(* IEC 61131-3 sources: SmartHomeNew/snapshots/2026-05-12, 47 files *)

(* ---- E_Heating_RootCause.dut ---- *)
TYPE E_Heating_RootCause :
(
    RC_NONE,
    RC_EMERGENCY_STOP,
    RC_GAS_SAFETY,
    RC_IO_OFFLINE,
    RC_BOILER_OFFLINE,
    RC_BOILER_ERROR,
    RC_NO_FLAME,
    RC_NO_FLOW,
    RC_PUMP_FAILURE,
    RC_VALVES_CLOSED,
    RC_NO_HEAT_TRANSFER,
    RC_LOW_SUPPLY_TEMP,
    RC_SENSOR_ERROR,
    RC_POLICY_BLOCKED,
    RC_UNKNOWN
);
END_TYPE

(* ---- E_Heating_Runtime_Phase.dut ---- *)
TYPE E_Heating_Runtime_Phase :
(
    HRP_DISABLED := 0,

    // Runtime startup / idle
    HRP_IDLE := 10,

    // Phase 1
    // DHW manager execution
    HRP_DHW := 20,

    // Phase 2
    // Heating runtime execution
    HRP_HEATING := 30,

    // Phase 3
    // Service and failsafe gating
    HRP_SERVICE_GATING := 40,

    // Phase 4
    // Runtime state publication
    HRP_STATE_PUBLICATION := 50,

    // Phase 5
    // Diagnostics / explainability
    HRP_DIAGNOSTICS := 60,

    // Phase 6
    // Output projection
    HRP_OUTPUT_PROJECTION := 70,

    // Runtime finished
    HRP_COMPLETE := 100,

    // Runtime error/fault state
    HRP_FAULT := 900
);
END_TYPE

(* ---- E_Modbus_RTU_RX_State.dut ---- *)
TYPE E_Modbus_RTU_RX_State :
(
    MB_RTU_RX_IDLE := 0,
    MB_RTU_RX_RECEIVING := 1,
    MB_RTU_RX_FRAME_READY := 2,
    MB_RTU_RX_CRC_ERROR := 3,
    MB_RTU_RX_OVERFLOW := 4,
    MB_RTU_RX_SHORT_FRAME := 5
);
END_TYPE

(* ---- E_System_Operating_Mode.dut ---- *)
TYPE E_System_Operating_Mode :
(
    MODE_NORMAL := 0,
    MODE_DEGRADED := 1,
    MODE_SAFE_STOP := 2,
    MODE_FREEZE_PROTECTION := 3
);
END_TYPE

(* ---- E_Trend_Parameter_Type.dut ---- *)
{attribute 'strict'}
TYPE E_Trend_Parameter_Type :
(
    TREND_PARAM_NONE := 0,
    TREND_PARAM_TEMP_AIR := 1,
    TREND_PARAM_TEMP_FLOOR := 2,
    TREND_PARAM_PRESSURE := 3,
    TREND_PARAM_PUMP_CURRENT := 4,
    TREND_PARAM_GAS_METHANE := 5,
    TREND_PARAM_GAS_CO := 6
) USINT;
END_TYPE

(* ---- ST_Device_Health.dut ---- *)
{attribute 'pack_mode' := '1'}
TYPE ST_Device_Health :
STRUCT
    Health_Score : BYTE := 100;
    Total_Runtime_Hours : UDINT;
    Starts_Count : UDINT;
    Last_Start_Current : REAL;
    Avg_Start_Current : REAL;
    Sample_Count : UDINT;
    Current_Sum : REAL;
    Maintenance_Required : BOOL;
    Warning_Message : STRING(50);
END_STRUCT
END_TYPE

(* ---- ST_FloorHeating_Circuit_Config.dut ---- *)
{attribute 'pack_mode' := '1'}
TYPE ST_FloorHeating_Circuit_Config :
STRUCT
    circuit_id : BYTE := 0;
    zone : BYTE := 0;
    manifold_id : BYTE := 1; // ID коллектора, к которому подключен контур
    sensor_id : BYTE := 1; // ID датчика температуры
    valve_id : BYTE := 1; // ID клапана
    control_type : BYTE := 1; // 0: по полу, 1: по воздуху
    design_temp : REAL := 35.0;
    min_temp : REAL := 20.0;
    max_temp : REAL := 45.0;
    pid_kp : REAL := 2.0;
    pwm_period_s : UINT := 600; // Период ШИМ в секундах (по умолчанию 10 минут)
END_STRUCT
END_TYPE

(* ---- ST_Heating_Runtime_Causality_Node.dut ---- *)
TYPE ST_Heating_Runtime_Causality_Node :
STRUCT
    // ======================================================
    // Node identity
    // ======================================================
    Node_ID : UINT;
    Node_Active : BOOL;

    // ======================================================
    // Runtime source state
    // ======================================================
    Runtime_Degraded : BOOL;
    Runtime_Fault : BOOL;

    // ======================================================
    // Cascade source state
    // ======================================================
    Cascade_Degraded : BOOL;
    Cascade_Boiler_Loss : BOOL;

    // ======================================================
    // OpenTherm source state
    // ======================================================
    OpenTherm_Degraded : BOOL;
    OpenTherm_Command_Invalid : BOOL;

    // ======================================================
    // Diagnostics source state
    // ======================================================
    Diagnostics_Degraded : BOOL;
    Explainability_Degraded : BOOL;

    // ======================================================
    // Sequencing/integrity state
    // ======================================================
    Sequencing_Invalid : BOOL;
    Ownership_Invalid : BOOL;
    Synchronization_Invalid : BOOL;

    // ======================================================
    // Causality severity
    // ======================================================
    Severity_Level : UINT;
    Root_Cause_Candidate : BOOL;

    // ======================================================
    // Node status
    // ======================================================
    Status_Code : UINT;
    Status_Text : STRING(128);
END_STRUCT
END_TYPE

(* ---- ST_Heating_Runtime_Execution_Frame.dut ---- *)
TYPE ST_Heating_Runtime_Execution_Frame :
STRUCT
    // ======================================================
    // Execution phase
    // ======================================================
    Phase : E_Heating_Runtime_Phase;

    // ======================================================
    // Execution lifecycle
    // ======================================================
    Frame_Started : BOOL;
    Frame_Completed : BOOL;
    Frame_Failed : BOOL;

    // ======================================================
    // Execution timing
    // ======================================================
    Frame_Start_MS : UDINT;
    Frame_End_MS : UDINT;
    Frame_Duration_MS : UDINT;

    // ======================================================
    // Execution integrity
    // ======================================================
    Sequencing_Valid : BOOL;
    Ownership_Valid : BOOL;
    Synchronization_Valid : BOOL;

    // ======================================================
    // Execution telemetry
    // ======================================================
    Runtime_Jitter_Detected : BOOL;
    Runtime_Latency_Detected : BOOL;
    Runtime_Degraded : BOOL;

    // ======================================================
    // Execution status
    // ======================================================
    Status_Code : UINT;
    Status_Text : STRING(128);
END_STRUCT
END_TYPE

(* ---- ST_Heating_Schedule_Event.dut ---- *)
{attribute 'pack_mode' := '1'}
TYPE ST_Heating_Schedule_Event :
STRUCT
    Enabled : BOOL := FALSE;
    Comfort_Time_MS : UDINT := 28800000; // 08:00 from midnight
    Weekday_Mask : BYTE := 127; // bit0=Mon ... bit6=Sun
    Preheat_Boost : REAL := 0.5;
    Adaptive_Enabled : BOOL := TRUE;
    Adaptive_Step_MS : UDINT := 300000; // 5 min
    Adaptive_Max_Offset_MS : UDINT := 3600000; // 60 min
END_STRUCT
END_TYPE

(* ---- ST_Modbus_RTU_Config.dut ---- *)
TYPE ST_Modbus_RTU_Config :
STRUCT
    Port_Name : STRING(32);
    Baudrate : UDINT;
    Parity : BYTE; // 0=None, 1=Even, 2=Odd
    Stop_Bits : BYTE; // 1 or 2
    Data_Bits : BYTE; // usually 8
    Slave_ID : BYTE;
    Poll_Interval_MS : UDINT;
    Request_Timeout_MS : UDINT;
    Retry_Count : INT;
END_STRUCT
END_TYPE

(* ---- ST_Modbus_RTU_Frame.dut ---- *)
TYPE ST_Modbus_RTU_Frame :
STRUCT
    Valid : BOOL;
    Length : UINT;
    Data : ARRAY[0..255] OF BYTE;
    CRC : WORD;
END_STRUCT
END_TYPE

(* ---- ST_OpenTherm_Register_Map.dut ---- *)
TYPE ST_OpenTherm_Register_Map :
STRUCT
    // Register offsets inside one boiler adapter block.
    // Real Modbus device addressing is configured by Base_Register + offsets.
    Base_Register : UINT;
    Cmd_Enable_Offset : UINT;
    Cmd_Setpoint_x10_Offset : UINT;
    Cmd_Seq_Lo_Offset : UINT;
    Cmd_Seq_Hi_Offset : UINT;

    Status_Heartbeat_Lo_Offset : UINT;
    Status_Heartbeat_Hi_Offset : UINT;
    Status_Ack_Seq_Lo_Offset : UINT;
    Status_Ack_Seq_Hi_Offset : UINT;
    Status_Word_Offset : UINT;
    Error_Code_Offset : UINT;
    Modulation_x10_Offset : UINT;
    Boiler_Temp_x10_Offset : UINT;
END_STRUCT
END_TYPE

(* ---- GVL_ACCESS_OUTPUT.gvl ---- *)
VAR_GLOBAL
    DO_Lock_1_Open : BOOL := FALSE;
    DO_Lock_1_Close : BOOL := FALSE;
    DO_Lock_2_Open : BOOL := FALSE;
    DO_Lock_2_Close : BOOL := FALSE;
    DO_Gate_Open : BOOL := FALSE;
    DO_Wicket_Open : BOOL := FALSE;
END_VAR

(* ---- GVL_DIAGNOSTICS_EXT.gvl ---- *)
{attribute 'qualified_only'}
VAR_GLOBAL
    // Health scores (0..1)
    G_Health_Heating : REAL := 1.0;
    G_Health_Safety : REAL := 1.0;
    G_Health_IO : REAL := 1.0;

    // Error counters
    G_Error_Count_Heating : UDINT := 0;
    G_Error_Count_Safety : UDINT := 0;
    G_Error_Count_IO : UDINT := 0;

    // Last error timestamps
    G_Last_Error_Time_Heating : UDINT := 0;
    G_Last_Error_Time_Safety : UDINT := 0;
    G_Last_Error_Time_IO : UDINT := 0;

    // Timing
    G_Last_Update_Time : UDINT := 0;

    // Cycle / watchdog statistics (interval between diagnostics executions)
    G_Cycle_Expected_MS : UDINT := 250;
    G_Cycle_Warning_MS : UDINT := 375;
    G_Cycle_Critical_MS : UDINT := 500;
    G_Cycle_Last_MS : UDINT := 0;
    G_Cycle_Max_MS : UDINT := 0;
    G_Cycle_Min_MS : UDINT := 0;
    G_Cycle_Avg_MS : REAL := 0.0;
    G_Cycle_Sample_Count : UDINT := 0;
    G_Cycle_Overrun_Count : UDINT := 0;
    G_Cycle_Critical_Count : UDINT := 0;
    G_Cycle_Last_Overrun_MS : UDINT := 0;
    G_Cycle_Last_Overrun_Time_MS : UDINT := 0;
    G_Cycle_Overrun_Active : BOOL := FALSE;
    G_Cycle_Critical_Active : BOOL := FALSE;

    // States
    G_Heating_State : INT := 0; // 0=OK,1=DEGRADED,2=CRITICAL
    G_Safety_State : INT := 0;
    G_IO_State : INT := 0;
END_VAR

(* ---- GVL_HEATING_REQUEST.gvl ---- *)
VAR_GLOBAL
    G_Freeze_Request : BOOL := FALSE;
    G_Target_Temperature : REAL := 0.0;
    G_Preheat_Request : BOOL := FALSE;
END_VAR

(* ---- GVL_INTENT_POLICY.gvl ---- *)
{attribute 'qualified_only'}
VAR_GLOBAL
    // Policy intent signals (NO logic, only transport)

    G_Preheat_Request : BOOL;
    G_Freeze_Request : BOOL;
    G_Eco_Mode_Request : BOOL;

    // Zone-level intents
    G_Zone_Heating_Request : ARRAY[1..GVL_CONSTANTS.C_MAX_ZONES] OF BOOL;
    G_Zone_Target_Adjustment : ARRAY[1..GVL_CONSTANTS.C_MAX_ZONES] OF REAL;

END_VAR

(* ---- GVL_SCENARIO_CONFIG.gvl ---- *)
{attribute 'qualified_only'}
VAR_GLOBAL
    // Scenario Engine configuration.
    // Used by PRG_Scenario_Engine only.

    G_Night_Start_Hour : INT := 22;
    G_Night_End_Hour : INT := 6;
    G_Access_Secure_Start_Hour : INT := 23;
    G_Access_Secure_End_Hour : INT := 5;

    G_Comfort_Base_Score : REAL := 10.0;
    G_Night_Base_Score : REAL := 40.0;
    G_Preheat_Base_Score : REAL := 50.0;
    G_VentBoost_Base_Score : REAL := 45.0;
    G_AccessSecure_Base_Score : REAL := 30.0;

    G_VentBoost_Humidity_Threshold : REAL := 65.0;

    G_Night_Activation_Threshold : INT := 30;
    G_Comfort_Activation_Threshold : INT := 40;
    G_VentBoost_Activation_Threshold : INT := 40;
    G_AccessSecure_Activation_Threshold : INT := 25;

    G_Fallback_Adapt_Confidence : REAL := 0.5;
    G_Fallback_Input_Confidence : REAL := 0.5;
END_VAR

(* ---- GVL_WATER_OUTPUT.gvl ---- *)
VAR_GLOBAL
    DO_Water_Valve_35_Close : BOOL := FALSE;
    DO_Water_Valve_36_Close : BOOL := FALSE;
    DO_Water_Zone_Enable : ARRAY[1..GVL_CONSTANTS.C_MAX_WATER_ZONES] OF BOOL;
END_VAR

(* ---- FB_Access_Control.st ---- *)
FUNCTION_BLOCK FB_Access_Control
VAR_INPUT
    VI_System_Time_MS   : UDINT; // Системное время (мс)
    VI_IsActivePLC      : BOOL; // Флаг: Данный ПЛК является ведущим (Active)
    VI_Armed            : BOOL; // Статус: Система безопасности находится под охраной
    VI_System_Mode      : E_System_Operating_Mode; // Агрегированный режим работы системы

    // Команды управления от HMI (через GVL_CONFIG)
    VI_Gate_Open_Req    : BOOL; // Запрос пользователя на открытие въездных ворот
    VI_Wicket_Open_Req  : BOOL; // Запрос пользователя на открытие калитки
    VI_Lock_1_Open_Req  : BOOL; // Запрос на разблокировку основного электрозамка дома
    VI_Lock_1_Close_Req : BOOL; // Запрос на блокировку основного электрозамка дома
    VI_Lock_2_Open_Req  : BOOL; // Запрос на разблокировку дополнительного электрозамка
    VI_Lock_2_Close_Req : BOOL; // Запрос на блокировку дополнительного электрозамка

    // Авторизация
    VI_PIN_Code         : STRING(4); // ПИН-код для авторизации
    VI_RFID_Tag         : STRING(20); // RFID/NFC метка для авторизации

    // Настройки из конфигурации безопасности (длительности импульсов)
    VI_Config           : ST_Security_Global_Config;
END_VAR
VAR_IN_OUT
    VI_Access_Codes     : ARRAY[1..GVL_CONSTANTS.C_MAX_ACCESS_CODES] OF DWORD;
    VI_RFID_Tags        : ARRAY[1..GVL_CONSTANTS.C_MAX_ACCESS_CODES] OF STRING(20);
END_VAR
VAR_OUTPUT
    VO_Gate_Open        : BOOL; // Выход: Импульс на открытие ворот (сухой контакт)
    VO_Wicket_Open      : BOOL; // Выход: Импульс на открытие калитки (электрозащелка)
    VO_Lock_1_Open      : BOOL; // Выход: Импульс на разблокировку замка №1
    VO_Lock_1_Close     : BOOL; // Выход: Импульс на блокировку замка №1
    VO_Lock_2_Open      : BOOL; // Выход: Импульс на разблокировку замка №2
    VO_Lock_2_Close     : BOOL; // Выход: Импульс на блокировку замка №2
END_VAR
VAR
    // Таймеры для формирования импульсов управления заданной длительности
    L_Gate_Timer        : TP; // Таймер импульса ворот
    L_Wicket_Timer      : TP; // Таймер импульса калитки
    L_Lock_1_Open_T     : TP; // Таймер открытия замка №1
    L_Lock_1_Close_T    : TP; // Таймер закрытия замка №1
    L_Lock_2_Open_T     : TP; // Таймер открытия замка №2
    L_Lock_2_Close_T    : TP; // Таймер закрытия замка №2

    L_Prev_Armed        : BOOL; // Предыдущее состояние охраны (для детекции фронта постановки)
    L_Auto_Lock_Req     : BOOL; // Флаг автоматического закрытия всех замков при постановке на охрану

    R_Trig_Gate         : R_TRIG;
    R_Trig_Wicket       : R_TRIG;
    R_Trig_Lock_1_O     : R_TRIG;
    R_Trig_Lock_1_C     : R_TRIG;
    R_Trig_Lock_2_O     : R_TRIG;
    R_Trig_Lock_2_C     : R_TRIG;

    fbAccessCode        : FB_AccessCode_Manager;
    L_Valid_PIN         : BOOL;
END_VAR

// Если ПЛК находится в режиме Standby (резерв), он не должен управлять выходами
IF NOT VI_IsActivePLC THEN
    RETURN;
END_IF;

IF VI_System_Mode = E_System_Operating_Mode.MODE_SAFE_STOP THEN
    VO_Gate_Open := FALSE;
    VO_Wicket_Open := FALSE;
    VO_Lock_1_Open := FALSE;
    VO_Lock_2_Open := FALSE;
    RETURN;
END_IF;

// 1. Логика автоматического закрытия замков при постановке на охрану (ТЗ 3.0)
// При переходе системы в режим "Охрана" принудительно блокируем все замки
IF VI_Armed AND NOT L_Prev_Armed THEN
    L_Auto_Lock_Req := TRUE;
END_IF;
L_Prev_Armed := VI_Armed;

// Детекторы фронта для команд
R_Trig_Gate(CLK := VI_Gate_Open_Req);
R_Trig_Wicket(CLK := VI_Wicket_Open_Req);
R_Trig_Lock_1_O(CLK := VI_Lock_1_Open_Req);
R_Trig_Lock_1_C(CLK := VI_Lock_1_Close_Req OR L_Auto_Lock_Req);
R_Trig_Lock_2_O(CLK := VI_Lock_2_Open_Req);
R_Trig_Lock_2_C(CLK := VI_Lock_2_Close_Req OR L_Auto_Lock_Req);

// Проверка PIN-кода или RFID-метки через менеджер кодов
fbAccessCode(
    VI_System_Time_MS := VI_System_Time_MS,
    VI_IsActivePLC := VI_IsActivePLC,
    VI_Code_To_Check := VI_PIN_Code,
    VI_RFID_To_Check := VI_RFID_Tag,
    VI_Access_Codes := VI_Access_Codes,
    VI_RFID_Tags := VI_RFID_Tags,
    VO_Code_Valid => L_Valid_PIN
);

// 2. Формирование импульсов управления исполнительными механизмами (Pulse Control)
// Открытие ворот и калитки требует валидного ПИН-кода или RFID-метки, если система под охраной
L_Gate_Timer(IN := R_Trig_Gate.Q AND (NOT VI_Armed OR L_Valid_PIN), PT := TO_TIME(VI_Config.gate_open_pulse_ms));
VO_Gate_Open := L_Gate_Timer.Q;

L_Wicket_Timer(IN := R_Trig_Wicket.Q AND (NOT VI_Armed OR L_Valid_PIN), PT := TO_TIME(VI_Config.wicket_open_pulse_ms));
VO_Wicket_Open := L_Wicket_Timer.Q;

L_Lock_1_Open_T(IN := R_Trig_Lock_1_O.Q AND (NOT VI_Armed OR L_Valid_PIN), PT := TO_TIME(VI_Config.lock_open_pulse_ms));
VO_Lock_1_Open := L_Lock_1_Open_T.Q;

L_Lock_1_Close_T(IN := R_Trig_Lock_1_C.Q, PT := TO_TIME(VI_Config.lock_close_pulse_ms));
VO_Lock_1_Close := L_Lock_1_Close_T.Q;

L_Lock_2_Open_T(IN := R_Trig_Lock_2_O.Q AND (NOT VI_Armed OR L_Valid_PIN), PT := TO_TIME(VI_Config.lock_open_pulse_ms));
VO_Lock_2_Open := L_Lock_2_Open_T.Q;

L_Lock_2_Close_T(IN := R_Trig_Lock_2_C.Q, PT := TO_TIME(VI_Config.lock_close_pulse_ms));
VO_Lock_2_Close := L_Lock_2_Close_T.Q;

// Сброс флага автоматического закрытия
IF L_Auto_Lock_Req THEN
    L_Auto_Lock_Req := FALSE;
END_IF;
// >>> BULK_SYNC_ANCHOR: FB_Access_Control <<<
END_FUNCTION_BLOCK

(* ---- FB_AccessCode_Manager.st ---- *)
FUNCTION_BLOCK FB_AccessCode_Manager
VAR_INPUT
    VI_System_Time_MS : UDINT;
    VI_IsActivePLC    : BOOL;
    VI_Code_To_Check  : STRING(4);
    VI_RFID_To_Check  : STRING(20);
END_VAR
VAR_IN_OUT
    VI_Access_Codes   : ARRAY[1..GVL_CONSTANTS.C_MAX_ACCESS_CODES] OF DWORD;
    VI_RFID_Tags      : ARRAY[1..GVL_CONSTANTS.C_MAX_ACCESS_CODES] OF STRING(20);
END_VAR
VAR_OUTPUT
    VO_Code_Valid     : BOOL;
END_VAR
VAR
    L_i : INT;
    pCode : POINTER TO BYTE;
    L_CRC_Calc : FB_CRC32_Calculator;
    L_Input_Hash : DWORD;
END_VAR

VO_Code_Valid := FALSE;

// Вычисляем хэш введенного кода
IF LEN(VI_Code_To_Check) > 0 THEN
    pCode := ADR(VI_Code_To_Check);
    L_Input_Hash := 0;
    FOR L_i := 1 TO GVL_CONSTANTS.C_MAX_ACCESS_CODES DO
        IF VI_Access_Codes[L_i] <> 0 AND VI_Access_Codes[L_i] = L_Input_Hash THEN
            VO_Code_Valid := TRUE;
            RETURN;
        END_IF;
    END_FOR;
END_IF;

// Проверяем RFID метку
IF LEN(VI_RFID_To_Check) > 0 THEN
    FOR L_i := 1 TO GVL_CONSTANTS.C_MAX_ACCESS_CODES DO
        IF VI_RFID_Tags[L_i] <> '' AND VI_RFID_Tags[L_i] = VI_RFID_To_Check THEN
            VO_Code_Valid := TRUE;
            RETURN;
        END_IF;
    END_FOR;
END_IF;
// >>> BULK_SYNC_ANCHOR: FB_AccessCode_Manager <<<
END_FUNCTION_BLOCK

(* ---- FB_Command_Deduplication.st ---- *)
FUNCTION_BLOCK FB_Command_Deduplication
VAR_INPUT
    VI_Command_ID : UDINT; // Unique ID from Gateway/HMI
    VI_Command_Type : E_Gateway_Command_Type;
    VI_Command_Value : REAL;
    VI_System_Time_MS : UDINT;
END_VAR
VAR_OUTPUT
    VO_Is_New_Command : BOOL; // TRUE if this command should be executed
    VO_Processed_ID : UDINT;
END_VAR
VAR
    L_Processed_History : ARRAY[0..GVL_CONSTANTS.C_MAX_DEDUPLICATION_HISTORY-1] OF UDINT; // Ring buffer of last processed IDs
    L_Processed_Times   : ARRAY[0..GVL_CONSTANTS.C_MAX_DEDUPLICATION_HISTORY-1] OF UDINT; // Timestamps for processed IDs
    L_History_Index : INT := 0;
    L_i : INT;
    L_Found : BOOL;
END_VAR

// Check if command ID is already in history
L_Found := FALSE;
FOR L_i := 0 TO GVL_CONSTANTS.C_MAX_DEDUPLICATION_HISTORY-1 DO
    IF L_Processed_History[L_i] = VI_Command_ID AND VI_Command_ID <> 0 THEN
        // Check if the command is not too old (e.g., 1 hour = 3600000 ms)
        IF (VI_System_Time_MS - L_Processed_Times[L_i]) < 3600000 THEN
            L_Found := TRUE;
            EXIT;
        END_IF;
    END_IF;
END_FOR;

IF NOT L_Found AND VI_Command_ID <> 0 THEN
    // New command detected
    VO_Is_New_Command := TRUE;
    VO_Processed_ID := VI_Command_ID;

    // Add to history
    L_Processed_History[L_History_Index] := VI_Command_ID;
    L_Processed_Times[L_History_Index] := VI_System_Time_MS;
    L_History_Index := L_History_Index + 1;
    IF L_History_Index > GVL_CONSTANTS.C_MAX_DEDUPLICATION_HISTORY-1 THEN
        L_History_Index := 0;
    END_IF;
ELSE
    // Duplicate or empty command
    VO_Is_New_Command := FALSE;
    VO_Processed_ID := 0;
END_IF;
END_FUNCTION_BLOCK

(* ---- FB_Heating_Adaptive_Target.st ---- *)
// ==============================================================================
// Adaptive target calculation for heating supply temperature
// ==============================================================================
FUNCTION_BLOCK FB_Heating_Adaptive_Target
VAR_INPUT
    VI_Base_Target_Supply_Temp : REAL;
    VI_Global_Target_Temperature : REAL;
END_VAR

VAR_IN_OUT
    VI_Zone_Configs : ARRAY[1..GVL_CONSTANTS.C_MAX_HEATING_CIRCUITS] OF ST_FloorHeating_Circuit_Config;
    VI_Floor_Temps : ARRAY[1..GVL_CONSTANTS.C_MAX_HEATING_CIRCUITS] OF REAL;
    VI_Room_Temps : ARRAY[1..GVL_CONSTANTS.C_MAX_ZONES] OF REAL;
END_VAR

VAR_OUTPUT
    VO_Target_Supply_Temp : REAL;
    VO_Adaptive_Correction : REAL;
    VO_Adaptive_Effective_Delta : REAL;
    VO_Adaptive_Max_Delta : REAL;
END_VAR

VAR
    L_Adaptive_Zone_i : INT;
    L_Zone_Index : INT;
    L_Adaptive_Delta : REAL;
    L_Adaptive_Weighted_Sum : REAL;
    L_Adaptive_Weight_Total : REAL;
    L_Adaptive_Weight : REAL;
END_VAR

VO_Target_Supply_Temp := VI_Base_Target_Supply_Temp;
VO_Adaptive_Max_Delta := 0.0;
L_Adaptive_Weighted_Sum := 0.0;
L_Adaptive_Weight_Total := 0.0;
VO_Adaptive_Effective_Delta := 0.0;
VO_Adaptive_Correction := 0.0;

IF VI_Global_Target_Temperature > 0.0 THEN
    VO_Target_Supply_Temp := VI_Global_Target_Temperature;
END_IF;

FOR L_Adaptive_Zone_i := 1 TO GVL_CONSTANTS.C_MAX_HEATING_CIRCUITS DO
    L_Zone_Index := VI_Zone_Configs[L_Adaptive_Zone_i].zone;

    IF (L_Zone_Index >= 1) AND (L_Zone_Index <= GVL_CONSTANTS.C_MAX_ZONES) THEN
        CASE VI_Zone_Configs[L_Adaptive_Zone_i].control_type OF
            0:
                L_Adaptive_Delta :=
                    VI_Zone_Configs[L_Adaptive_Zone_i].design_temp -
                    VI_Floor_Temps[L_Adaptive_Zone_i];
                L_Adaptive_Weight := 0.6;
            1, 2:
                L_Adaptive_Delta :=
                    VI_Zone_Configs[L_Adaptive_Zone_i].design_temp -
                    VI_Room_Temps[L_Zone_Index];
                L_Adaptive_Weight := 1.0;
            ELSE
                L_Adaptive_Delta :=
                    VI_Zone_Configs[L_Adaptive_Zone_i].design_temp -
                    VI_Room_Temps[L_Zone_Index];
                L_Adaptive_Weight := 0.8;
        END_CASE;

        IF L_Zone_Index <= 4 THEN
            L_Adaptive_Weight := L_Adaptive_Weight * 1.2;
        ELSIF L_Zone_Index >= 9 THEN
            L_Adaptive_Weight := L_Adaptive_Weight * 0.7;
        END_IF;

        IF L_Adaptive_Weight > 2.0 THEN
            L_Adaptive_Weight := 2.0;
        ELSIF L_Adaptive_Weight < 0.2 THEN
            L_Adaptive_Weight := 0.2;
        END_IF;

        IF L_Adaptive_Delta > VO_Adaptive_Max_Delta THEN
            VO_Adaptive_Max_Delta := L_Adaptive_Delta;
        END_IF;

        L_Adaptive_Weighted_Sum := L_Adaptive_Weighted_Sum + (L_Adaptive_Delta * L_Adaptive_Weight);
        L_Adaptive_Weight_Total := L_Adaptive_Weight_Total + L_Adaptive_Weight;
    END_IF;
END_FOR;

IF L_Adaptive_Weight_Total > 0.0 THEN
    VO_Adaptive_Effective_Delta := L_Adaptive_Weighted_Sum / L_Adaptive_Weight_Total;
END_IF;

IF VO_Adaptive_Effective_Delta > 1.5 THEN
    VO_Adaptive_Correction := 2.0;
ELSIF VO_Adaptive_Effective_Delta > 0.7 THEN
    VO_Adaptive_Correction := 1.0;
ELSIF VO_Adaptive_Effective_Delta < -1.5 THEN
    VO_Adaptive_Correction := -2.0;
ELSIF VO_Adaptive_Effective_Delta < -0.7 THEN
    VO_Adaptive_Correction := -1.0;
ELSE
    VO_Adaptive_Correction := 0.0;
END_IF;

IF VO_Adaptive_Max_Delta > 2.5 AND VO_Adaptive_Correction < 2.0 THEN
    VO_Adaptive_Correction := 2.0;
END_IF;

VO_Target_Supply_Temp := VO_Target_Supply_Temp + VO_Adaptive_Correction;

IF VO_Target_Supply_Temp < 20.0 THEN
    VO_Target_Supply_Temp := 20.0;
ELSIF VO_Target_Supply_Temp > 45.0 THEN
    VO_Target_Supply_Temp := 45.0;
END_IF;

// >>> BULK_SYNC_ANCHOR: FB_Heating_Adaptive_Target <<<
END_FUNCTION_BLOCK

(* ---- FB_Heating_Allocation_Filter.st ---- *)
// ==============================================================================
// Heating allocation filter
// Runtime decision gate between Demand_Map and Manifold_Control.
//
// IMPORTANT:
// This FB is NOT a second runtime owner.
// This FB is NOT an orchestration layer.
//
// Actual ownership remains in:
// PRG_Heating
// → FB_Heating_System_Manager
// → active subsystem owners.
//
// Current responsibility:
// - manifold availability gating;
// - service-state filtering;
// - freeze-mode exceptions;
// - bounded demand authorization.
//
// Optional responsibility when explicitly enabled:
// - priority-based allocation;
// - thermal budget limiting.
// ==============================================================================
FUNCTION_BLOCK FB_Heating_Allocation_Filter
VAR_INPUT
    // Master runtime enable.
    // FALSE = strict passthrough.
    VI_Enable : BOOL;

    // Optional policy layer.
    // FALSE = only availability/service/degraded gate is active.
    VI_Enable_Policy_Allocation : BOOL := FALSE;

    // System-level context.
    VI_Freeze_Mode_Active : BOOL;
    VI_DHW_Heating_Demand : BOOL;

    // Current manifold demand.
    VI_Manifold_Demand_Map : ARRAY[1..GVL_CONSTANTS.C_MAX_MANIFOLDS] OF BOOL;

    // Runtime/service availability.
    VI_Manifold_Available : ARRAY[1..GVL_CONSTANTS.C_MAX_MANIFOLDS] OF BOOL;
    VI_Manifold_In_Service : ARRAY[1..GVL_CONSTANTS.C_MAX_MANIFOLDS] OF BOOL;
    VI_Manifold_Subsystem_Degraded : ARRAY[1..GVL_CONSTANTS.C_MAX_MANIFOLDS] OF BOOL;

    // Policy inputs from active configuration.
    VI_Manifold_Base_Priority : ARRAY[1..GVL_CONSTANTS.C_MAX_MANIFOLDS] OF INT;
    VI_Manifold_Thermal_Weight : ARRAY[1..GVL_CONSTANTS.C_MAX_MANIFOLDS] OF REAL;
    VI_Max_Thermal_Budget : REAL := REAL#0.0;
END_VAR
VAR_OUTPUT
    // Authorized demand.
    VO_Manifold_Demand_Filtered : ARRAY[1..GVL_CONSTANTS.C_MAX_MANIFOLDS] OF BOOL;

    // Runtime degraded indicator.
    VO_Allocation_Degraded : BOOL;

    // Explainability/diagnostics.
    VO_Manifold_Allowed : ARRAY[1..GVL_CONSTANTS.C_MAX_MANIFOLDS] OF BOOL;
    VO_Manifold_Block_Reason : ARRAY[1..GVL_CONSTANTS.C_MAX_MANIFOLDS] OF E_Heating_Allocation_Block_Reason;

    // Policy diagnostics.
    VO_Manifold_Priority_Effective : ARRAY[1..GVL_CONSTANTS.C_MAX_MANIFOLDS] OF INT;
    VO_Thermal_Budget_Used : REAL;
END_VAR
VAR
    L_i : INT;
    L_CurrentPriority : INT;
    L_MaxPriority : INT;
    L_Used : REAL;
    L_Weight : REAL;
    L_AnyPolicyBlock : BOOL;
END_VAR

// ======================================================
// DEFAULT STATE
// ======================================================
VO_Allocation_Degraded := FALSE;
VO_Thermal_Budget_Used := REAL#0.0;
L_AnyPolicyBlock := FALSE;

FOR L_i := 1 TO GVL_CONSTANTS.C_MAX_MANIFOLDS DO
    VO_Manifold_Demand_Filtered[L_i] := VI_Manifold_Demand_Map[L_i];
    VO_Manifold_Allowed[L_i] := TRUE;
    VO_Manifold_Block_Reason[L_i] := E_Heating_Allocation_Block_Reason.NONE;
    VO_Manifold_Priority_Effective[L_i] := VI_Manifold_Base_Priority[L_i];
END_FOR;

// ======================================================
// STRICT PASSTHROUGH MODE
// ======================================================
IF NOT VI_Enable THEN
    RETURN;
END_IF;

// ======================================================
// FREEZE EXCEPTION MODE
//
// Freeze protection has higher authority than
// service gating and policy throttling.
// ======================================================
IF VI_Freeze_Mode_Active THEN
    FOR L_i := 1 TO GVL_CONSTANTS.C_MAX_MANIFOLDS DO
        IF VI_Manifold_Demand_Map[L_i] THEN
            VO_Manifold_Block_Reason[L_i] := E_Heating_Allocation_Block_Reason.FREEZE_BYPASS;
        END_IF;
    END_FOR;
    RETURN;
END_IF;

// ======================================================
// DHW PRIORITY GATE
//
// Manifold_Control already owns DHW shutdown.
// Keep this filter transparent during DHW hold to avoid
// creating duplicate DHW authority here.
// ======================================================
IF VI_DHW_Heating_Demand THEN
    FOR L_i := 1 TO GVL_CONSTANTS.C_MAX_MANIFOLDS DO
        IF VI_Manifold_Demand_Map[L_i] THEN
            VO_Manifold_Block_Reason[L_i] := E_Heating_Allocation_Block_Reason.DHW_BYPASS;
        END_IF;
    END_FOR;
    RETURN;
END_IF;

// ======================================================
// MANIFOLD AUTHORIZATION FILTER
// ======================================================
FOR L_i := 1 TO GVL_CONSTANTS.C_MAX_MANIFOLDS DO

    IF NOT VI_Manifold_Available[L_i] THEN
        VO_Manifold_Allowed[L_i] := FALSE;
        VO_Manifold_Block_Reason[L_i] := E_Heating_Allocation_Block_Reason.PRESSURE_UNAVAILABLE;
    END_IF;

    IF NOT VI_Manifold_In_Service[L_i] THEN
        VO_Manifold_Allowed[L_i] := FALSE;
        VO_Manifold_Block_Reason[L_i] := E_Heating_Allocation_Block_Reason.SERVICE_DISABLED;
    END_IF;

    IF VI_Manifold_Subsystem_Degraded[L_i] THEN
        VO_Manifold_Allowed[L_i] := FALSE;
        VO_Manifold_Block_Reason[L_i] := E_Heating_Allocation_Block_Reason.PREDICTIVE_DEGRADED;
    END_IF;

    IF VI_Manifold_Demand_Map[L_i] AND NOT VO_Manifold_Allowed[L_i] THEN
        VO_Manifold_Demand_Filtered[L_i] := FALSE;
        VO_Allocation_Degraded := TRUE;
    END_IF;

END_FOR;

// ======================================================
// OPTIONAL POLICY LAYER
//
// This layer can only reduce demand that is already
// authorized by availability/service/degraded checks.
// It never creates new demand and never writes outputs.
// ======================================================
IF NOT VI_Enable_Policy_Allocation THEN
    RETURN;
END_IF;

// Invalid or unset budget means no policy throttling.
IF VI_Max_Thermal_Budget <= REAL#0.0 THEN
    RETURN;
END_IF;

// Rebuild output demand from allowed candidates only.
FOR L_i := 1 TO GVL_CONSTANTS.C_MAX_MANIFOLDS DO
    VO_Manifold_Demand_Filtered[L_i] := FALSE;
END_FOR;

L_MaxPriority := 0;
FOR L_i := 1 TO GVL_CONSTANTS.C_MAX_MANIFOLDS DO
    IF VI_Manifold_Demand_Map[L_i] AND VO_Manifold_Allowed[L_i] THEN
        IF VO_Manifold_Priority_Effective[L_i] > L_MaxPriority THEN
            L_MaxPriority := VO_Manifold_Priority_Effective[L_i];
        END_IF;
    END_IF;
END_FOR;

L_Used := REAL#0.0;

FOR L_CurrentPriority := L_MaxPriority TO 0 BY -1 DO
    FOR L_i := 1 TO GVL_CONSTANTS.C_MAX_MANIFOLDS DO
        IF VI_Manifold_Demand_Map[L_i]
           AND VO_Manifold_Allowed[L_i]
           AND (VO_Manifold_Priority_Effective[L_i] = L_CurrentPriority) THEN

            L_Weight := VI_Manifold_Thermal_Weight[L_i];
            IF L_Weight <= REAL#0.0 THEN
                L_Weight := REAL#1.0;
            END_IF;

            IF (L_Used + L_Weight) <= VI_Max_Thermal_Budget THEN
                VO_Manifold_Demand_Filtered[L_i] := TRUE;
                L_Used := L_Used + L_Weight;
            ELSE
                L_AnyPolicyBlock := TRUE;
                IF VO_Manifold_Block_Reason[L_i] = E_Heating_Allocation_Block_Reason.NONE THEN
                    VO_Manifold_Block_Reason[L_i] := E_Heating_Allocation_Block_Reason.POLICY_BUDGET_SHED;
                END_IF;
            END_IF;
        END_IF;
    END_FOR;
END_FOR;

VO_Thermal_Budget_Used := L_Used;

IF L_AnyPolicyBlock THEN
    VO_Allocation_Degraded := TRUE;
END_IF;

END_FUNCTION_BLOCK
// >>> BULK_SYNC_ANCHOR: FB_Heating_Allocation_Filter <<<

(* ---- FB_Heating_Boiler_Control.st ---- *)
// ==============================================================================
// Heating boiler control helper
// ==============================================================================
FUNCTION_BLOCK FB_Heating_Boiler_Control
VAR_INPUT
    VI_System_Time_MS : UDINT;
    VI_IsActivePLC : BOOL;
    VI_DHW_Heating_Demand : BOOL;
    VI_DHW_Target_Temp : REAL;
    VI_Target_Supply_Temp : REAL;
    VI_Freeze_Mode_Active : BOOL;
    VI_Policy_Degraded : BOOL;
    VI_Manifold_Pumps : ARRAY[1..GVL_CONSTANTS.C_MAX_MANIFOLDS] OF BOOL;
    VI_Manifold_Valves : ARRAY[1..GVL_CONSTANTS.C_MAX_MANIFOLDS] OF REAL;
    VI_Boiler_Flame_Status : ARRAY[1..GVL_CONSTANTS.C_MAX_BOILERS] OF BOOL;
    VI_Boiler_Error_Status : ARRAY[1..GVL_CONSTANTS.C_MAX_BOILERS] OF BOOL;
    VI_Boiler_OT_Online : ARRAY[1..GVL_CONSTANTS.C_MAX_BOILERS] OF BOOL;
END_VAR
VAR_IN_OUT
    VI_Boiler_Modulation : ARRAY[1..GVL_CONSTANTS.C_MAX_BOILERS] OF REAL;
END_VAR
VAR_OUTPUT
    VO_Boiler_OT_Enable : ARRAY[1..GVL_CONSTANTS.C_MAX_BOILERS] OF BOOL;
    VO_Boiler_OT_Setpoint : ARRAY[1..GVL_CONSTANTS.C_MAX_BOILERS] OF REAL;
    VO_Boiler_Status : ARRAY[1..GVL_CONSTANTS.C_MAX_BOILERS] OF ST_Boiler_Status;
    VO_Any_Subsystem_Degraded : BOOL;
    VO_Lead_Boiler : BYTE;
    VO_Demand_Power : REAL;
END_VAR
VAR
    L_i : INT;
    L_Delta_MS : UDINT;
    L_Last_Scan_Time : UDINT;
    L_Scan_Time_Init : BOOL := FALSE;
    L_Boiler_Request_Enable : ARRAY[1..GVL_CONSTANTS.C_MAX_BOILERS] OF BOOL;
    L_Boiler_Request_Setpoint : ARRAY[1..GVL_CONSTANTS.C_MAX_BOILERS] OF REAL;
    L_Boiler_OT_Command_Valid : ARRAY[1..GVL_CONSTANTS.C_MAX_BOILERS] OF BOOL;
    L_Transport_Degraded : BOOL;
    L_Available_Count : UINT;
    L_Active_Count : UINT;
    L_Any_Transport_Degraded : BOOL;
    L_Any_Ignition_Timeout : BOOL;
    L_Any_Flame : BOOL;
    L_Boiler_Life : ARRAY[1..GVL_CONSTANTS.C_MAX_BOILERS] OF FB_Lifetime_Predictor;
    fbBoilerCascade : FB_Boiler_Cascade_Manager;
    fbBoilerOpenTherm : FB_Boiler_OpenTherm_Interface;
END_VAR

VO_Any_Subsystem_Degraded := FALSE;
VO_Demand_Power := 0.0;

L_Available_Count := 0;
L_Active_Count := 0;
L_Any_Transport_Degraded := FALSE;
L_Any_Ignition_Timeout := FALSE;
L_Any_Flame := FALSE;

FOR L_i := 1 TO GVL_CONSTANTS.C_MAX_MANIFOLDS DO
    IF VI_Manifold_Pumps[L_i] THEN
        VO_Demand_Power := VO_Demand_Power + VI_Manifold_Valves[L_i];
    END_IF;
END_FOR;

IF VI_Freeze_Mode_Active AND VO_Demand_Power < 20.0 THEN
    VO_Demand_Power := 20.0;
END_IF;

IF VI_Policy_Degraded THEN
    IF VO_Demand_Power > 60.0 THEN
        VO_Demand_Power := 60.0;
    END_IF;
END_IF;

fbBoilerCascade(
    VI_Enable := VI_IsActivePLC AND ((VO_Demand_Power > GVL_CONSTANTS.C_BOILER_CASCADE_MIN_DEMAND) OR VI_Freeze_Mode_Active OR VI_DHW_Heating_Demand),
    VI_System_Time_MS := VI_System_Time_MS,
    VI_Boiler_Stop := FALSE,
    VI_DHW_Heating_Demand := VI_DHW_Heating_Demand,
    VI_DHW_Target_Temp := VI_DHW_Target_Temp,
    VI_Target_Supply_Temp := VI_Target_Supply_Temp,
    VI_Demand_Power := VO_Demand_Power,
    VI_Boiler_Flame_Status := VI_Boiler_Flame_Status,
    VI_Boiler_Error_Status := VI_Boiler_Error_Status,
    VI_Boiler_OT_Online := VI_Boiler_OT_Online,
    VI_Boiler_Modulation := VI_Boiler_Modulation,
    VO_Boiler_Enable => L_Boiler_Request_Enable,
    VO_Boiler_Setpoint => L_Boiler_Request_Setpoint,
    VO_Lead_Boiler => VO_Lead_Boiler
);

FOR L_i := 1 TO GVL_CONSTANTS.C_MAX_BOILERS DO
    IF L_Boiler_Request_Enable[L_i] THEN
        L_Boiler_Request_Setpoint[L_i] := LIMIT(
            GVL_CONSTANTS.C_BOILER_SETPOINT_MIN,
            L_Boiler_Request_Setpoint[L_i],
            80.0
        );
    END_IF;
END_FOR;

FOR L_i := 1 TO GVL_CONSTANTS.C_MAX_BOILERS DO
    IF NOT VI_Boiler_OT_Online[L_i] OR VI_Boiler_Error_Status[L_i] THEN
        L_Boiler_Request_Enable[L_i] := FALSE;
        L_Boiler_Request_Setpoint[L_i] := 0.0;
    END_IF;
END_FOR;

fbBoilerOpenTherm(
    VI_Enable := L_Boiler_Request_Enable,
    VI_Setpoint := L_Boiler_Request_Setpoint,
    VI_OT_Online := VI_Boiler_OT_Online,
    VI_OT_Error := VI_Boiler_Error_Status,
    VO_OT_Enable => VO_Boiler_OT_Enable,
    VO_OT_Setpoint => VO_Boiler_OT_Setpoint,
    VO_OT_Command_Valid => L_Boiler_OT_Command_Valid
);

FOR L_i := 1 TO GVL_CONSTANTS.C_MAX_BOILERS DO

    L_Transport_Degraded :=
        L_Boiler_Request_Enable[L_i] AND
        (
            NOT L_Boiler_OT_Command_Valid[L_i] OR
            NOT VI_Boiler_OT_Online[L_i] OR
            VI_Boiler_Error_Status[L_i]
        );

    VO_Boiler_Status[L_i].OT_Online := VI_Boiler_OT_Online[L_i];
    VO_Boiler_Status[L_i].OT_Command_Valid := L_Boiler_OT_Command_Valid[L_i];
    VO_Boiler_Status[L_i].OT_Transport_Degraded := L_Transport_Degraded;
    VO_Boiler_Status[L_i].OT_Adapter_Error :=
        GVL_OPENTHERM_ADAPTER.G_Status[L_i].Adapter_Error;

    VO_Boiler_Status[L_i].Active := L_Boiler_Request_Enable[L_i];
    VO_Boiler_Status[L_i].Running := VI_Boiler_Flame_Status[L_i];
    VO_Boiler_Status[L_i].Warning := L_Transport_Degraded;
    VO_Boiler_Status[L_i].Error := VI_Boiler_Error_Status[L_i];

    VO_Boiler_Status[L_i].Available :=
        VI_Boiler_OT_Online[L_i] AND
        NOT VI_Boiler_Error_Status[L_i] AND
        NOT L_Transport_Degraded;

    VO_Boiler_Status[L_i].Selected_By_Cascade :=
        L_Boiler_Request_Enable[L_i];

    VO_Boiler_Status[L_i].Transport_Missing :=
        NOT VI_Boiler_OT_Online[L_i];

    VO_Boiler_Status[L_i].Flame_Missing :=
        L_Boiler_Request_Enable[L_i] AND
        NOT VI_Boiler_Flame_Status[L_i] AND
        NOT L_Transport_Degraded;

    VO_Boiler_Status[L_i].Ignition_Timeout :=
        VO_Boiler_Status[L_i].Flame_Missing AND
        (GVL_STATE.G_Boiler_OT_Command_Age_MS[L_i] > 30000);

    VO_Boiler_Status[L_i].Degraded :=
        L_Transport_Degraded OR
        VO_Boiler_Status[L_i].Ignition_Timeout;

    // ======================================================
    // CASCADE AGGREGATION
    // ======================================================
    IF VO_Boiler_Status[L_i].Available THEN
        L_Available_Count := L_Available_Count + 1;
    END_IF;

    IF VO_Boiler_Status[L_i].Selected_By_Cascade THEN
        L_Active_Count := L_Active_Count + 1;
    END_IF;

    IF VI_Boiler_Flame_Status[L_i] THEN
        L_Any_Flame := TRUE;
    END_IF;

    IF L_Transport_Degraded THEN
        L_Any_Transport_Degraded := TRUE;
    END_IF;

    IF VO_Boiler_Status[L_i].Ignition_Timeout THEN
        L_Any_Ignition_Timeout := TRUE;
    END_IF;

    IF VO_Boiler_Status[L_i].Degraded THEN
        VO_Any_Subsystem_Degraded := TRUE;
    END_IF;

END_FOR;

// ======================================================
// GLOBAL CASCADE SEMANTIC STATE
// ======================================================
GVL_STATE.G_Heating_Cascade_Active_Boilers := L_Active_Count;
GVL_STATE.G_Heating_Cascade_Available_Boilers := L_Available_Count;

GVL_STATE.G_Heating_Cascade_Available :=
    (L_Available_Count > 0);

GVL_STATE.G_Heating_Cascade_Partial_Capacity :=
    (L_Available_Count > 0) AND
    (L_Available_Count < GVL_CONSTANTS.C_MAX_BOILERS);

GVL_STATE.G_Heating_Cascade_Transport_Degraded :=
    L_Any_Transport_Degraded;

GVL_STATE.G_Heating_Cascade_Ignition_Timeout :=
    L_Any_Ignition_Timeout;

GVL_STATE.G_Heating_Cascade_No_Flame :=
    (L_Active_Count > 0) AND
    NOT L_Any_Flame;

GVL_STATE.G_Heating_Cascade_Degraded :=
    GVL_STATE.G_Heating_Cascade_Transport_Degraded OR
    GVL_STATE.G_Heating_Cascade_Ignition_Timeout OR
    GVL_STATE.G_Heating_Cascade_Partial_Capacity;

END_FUNCTION_BLOCK

(* ---- FB_Heating_Policy_Priority_Bridge.st ---- *)
// ==============================================================================
// Heating policy priority bridge
//
// Bounded mapper from advisory zone policy to manifold allocation priority.
//
// IMPORTANT:
// - does NOT own demand;
// - does NOT create demand;
// - does NOT control pumps/valves;
// - does NOT write outputs;
// - does NOT bypass safety or service gates.
//
// Responsibility:
// - map circuit->zone policy bias into manifold effective priority;
// - keep the result bounded and deterministic;
// - provide a safe input for FB_Heating_Allocation_Filter.
// ==============================================================================
FUNCTION_BLOCK FB_Heating_Policy_Priority_Bridge
VAR_INPUT
    VI_Enable : BOOL;

    VI_Zone_Valves : ARRAY[1..GVL_CONSTANTS.C_MAX_HEATING_CIRCUITS] OF BOOL;
    VI_Zone_Configs : ARRAY[1..GVL_CONSTANTS.C_MAX_HEATING_CIRCUITS] OF ST_FloorHeating_Circuit_Config;

    VI_Manifold_Base_Priority : ARRAY[1..GVL_CONSTANTS.C_MAX_MANIFOLDS] OF INT;
    VI_Zone_Priority_Bias : ARRAY[1..GVL_CONSTANTS.C_MAX_ZONES] OF REAL;
    VI_Policy_Priority_Multiplier : REAL;
END_VAR
VAR_OUTPUT
    VO_Manifold_Effective_Priority : ARRAY[1..GVL_CONSTANTS.C_MAX_MANIFOLDS] OF INT;
    VO_Manifold_Priority_Bias_Applied : ARRAY[1..GVL_CONSTANTS.C_MAX_MANIFOLDS] OF REAL;
    VO_Bridge_Active : BOOL;
END_VAR
VAR
    L_i : INT;
    L_Manifold_ID : INT;
    L_Zone_ID : INT;
    L_Multiplier : REAL;
    L_Bias : REAL;
    L_Score : REAL;
    L_MaxScore : ARRAY[1..GVL_CONSTANTS.C_MAX_MANIFOLDS] OF REAL;
    L_HasActiveCircuit : ARRAY[1..GVL_CONSTANTS.C_MAX_MANIFOLDS] OF BOOL;
END_VAR

// Default passthrough state.
VO_Bridge_Active := FALSE;

FOR L_i := 1 TO GVL_CONSTANTS.C_MAX_MANIFOLDS DO
    VO_Manifold_Effective_Priority[L_i] := VI_Manifold_Base_Priority[L_i];
    VO_Manifold_Priority_Bias_Applied[L_i] := REAL#1.0;
    L_MaxScore[L_i] := REAL#0.0;
    L_HasActiveCircuit[L_i] := FALSE;
END_FOR;

IF NOT VI_Enable THEN
    RETURN;
END_IF;

L_Multiplier := VI_Policy_Priority_Multiplier;
IF L_Multiplier <= REAL#0.0 THEN
    L_Multiplier := REAL#1.0;
ELSIF L_Multiplier < REAL#0.3 THEN
    L_Multiplier := REAL#0.3;
ELSIF L_Multiplier > REAL#1.0 THEN
    L_Multiplier := REAL#1.0;
END_IF;

IF ABS(L_Multiplier - REAL#1.0) > REAL#0.001 THEN
    VO_Bridge_Active := TRUE;
END_IF;

FOR L_i := 1 TO GVL_CONSTANTS.C_MAX_HEATING_CIRCUITS DO
    IF VI_Zone_Valves[L_i] THEN
        L_Manifold_ID := TO_INT(VI_Zone_Configs[L_i].manifold_id);
        L_Zone_ID := TO_INT(VI_Zone_Configs[L_i].zone);

        IF (L_Manifold_ID >= 1)
           AND (L_Manifold_ID <= GVL_CONSTANTS.C_MAX_MANIFOLDS)
           AND (L_Zone_ID >= 1)
           AND (L_Zone_ID <= GVL_CONSTANTS.C_MAX_ZONES) THEN

            L_Bias := VI_Zone_Priority_Bias[L_Zone_ID];
            IF L_Bias <= REAL#0.0 THEN
                // Uninitialized advisory bias is treated as neutral.
                L_Bias := REAL#1.0;
            ELSIF L_Bias < REAL#0.3 THEN
                L_Bias := REAL#0.3;
            ELSIF L_Bias > REAL#1.5 THEN
                L_Bias := REAL#1.5;
            END_IF;

            IF ABS(L_Bias - REAL#1.0) > REAL#0.001 THEN
                VO_Bridge_Active := TRUE;
            END_IF;

            IF L_Bias > VO_Manifold_Priority_Bias_Applied[L_Manifold_ID] THEN
                VO_Manifold_Priority_Bias_Applied[L_Manifold_ID] := L_Bias;
            END_IF;

            L_Score := TO_REAL(VI_Manifold_Base_Priority[L_Manifold_ID]) * L_Multiplier * L_Bias;

            IF L_Score > L_MaxScore[L_Manifold_ID] THEN
                L_MaxScore[L_Manifold_ID] := L_Score;
            END_IF;

            L_HasActiveCircuit[L_Manifold_ID] := TRUE;
        END_IF;
    END_IF;
END_FOR;

FOR L_i := 1 TO GVL_CONSTANTS.C_MAX_MANIFOLDS DO
    IF L_HasActiveCircuit[L_i] THEN
        IF L_MaxScore[L_i] >= REAL#3.5 THEN
            VO_Manifold_Effective_Priority[L_i] := 4;
        ELSIF L_MaxScore[L_i] >= REAL#2.5 THEN
            VO_Manifold_Effective_Priority[L_i] := 3;
        ELSIF L_MaxScore[L_i] >= REAL#1.5 THEN
            VO_Manifold_Effective_Priority[L_i] := 2;
        ELSIF L_MaxScore[L_i] >= REAL#0.5 THEN
            VO_Manifold_Effective_Priority[L_i] := 1;
        ELSE
            VO_Manifold_Effective_Priority[L_i] := 0;
        END_IF;
    ELSE
        VO_Manifold_Effective_Priority[L_i] := VI_Manifold_Base_Priority[L_i];
        VO_Manifold_Priority_Bias_Applied[L_i] := REAL#1.0;
    END_IF;
END_FOR;

END_FUNCTION_BLOCK
// >>> BULK_SYNC_ANCHOR: FB_Heating_Policy_Priority_Bridge <<<

(* ---- FB_Heating_Predictive_Controller.st ---- *)
FUNCTION_BLOCK FB_Heating_Predictive_Controller
VAR
    L_i : INT;
    L_Time_To_Heat : UDINT;
    L_Time_To_Comfort : UDINT;
    L_Now_TOD : UDINT;
END_VAR

// ==============================================================================
// Ownership note
// ------------------------------------------------------------------------------
// This block owns predictive preheat decision only.
// It does NOT modify thermal demand. Thermal demand is owned by
// FB_Heating_Thermal_Model and may be interpreted by downstream advisory layers.
// ==============================================================================

L_Now_TOD := GVL_TIME_SERVICE.G_Time_Of_Day_MS;

FOR L_i := 1 TO GVL_CONSTANTS.C_MAX_ZONES DO

    L_Time_To_Heat := GVL_HEATING_POLICY.G_Zone_Time_To_Heat_MS[L_i];
    L_Time_To_Comfort := GVL_HEATING_POLICY.G_Zone_Comfort_Time_MS[L_i];

    // Predictive preheat decision.
    IF GVL_HEATING_POLICY.G_Zone_Schedule_Enabled[L_i] THEN

        IF L_Time_To_Comfort > L_Now_TOD THEN
            IF (L_Time_To_Comfort - L_Now_TOD) <= L_Time_To_Heat THEN
                GVL_HEATING_POLICY.G_Zone_Preheat_Needed[L_i] := TRUE;
            ELSE
                GVL_HEATING_POLICY.G_Zone_Preheat_Needed[L_i] := FALSE;
            END_IF;
        END_IF;

    END_IF;

    // Confidence gating.
    IF GVL_HEATING_POLICY.G_Zone_Thermal_Model_Confidence[L_i] < 0.1 THEN
        GVL_HEATING_POLICY.G_Zone_Preheat_Needed[L_i] := FALSE;
    END_IF;

END_FOR;

END_FUNCTION_BLOCK

(* ---- FB_Heating_Runtime_Diagnostics_Phase.st ---- *)
// ==============================================================================
// Heating runtime diagnostics phase
// Owns diagnostics publication for heating runtime sequencing.
// Does NOT own heating control or output decisions.
// ==============================================================================
FUNCTION_BLOCK FB_Heating_Runtime_Diagnostics_Phase
VAR_INPUT
    VI_Enable : BOOL;
    VI_System_Time_MS : UDINT;
END_VAR
VAR_OUTPUT
    VO_Executed : BOOL;
    VO_Valid : BOOL;
END_VAR
VAR
    fbRootCauseDiagnostics : FB_Heating_RootCause_Diagnostics;
    fbDiagEventManager : FB_Diagnostics_Event_Manager;

    L_i : INT;
    L_Any_Heating_Device_OOS : BOOL;
    L_Critical_Fault : BOOL;
    L_Device_Text : STRING(200);
    L_Critical_Text : STRING(200);
    L_Event_Text : STRING(200);
    L_Add_Text : STRING(80);
END_VAR

VO_Executed := FALSE;
VO_Valid := FALSE;

IF NOT VI_Enable THEN
    RETURN;
END_IF;

// ======================================================
// ROOT CAUSE DIAGNOSTICS
// ======================================================
fbRootCauseDiagnostics(
    VI_Enable := TRUE
);

// ======================================================
// DEFAULTS
// ======================================================
L_Any_Heating_Device_OOS := FALSE;
L_Critical_Fault := FALSE;
L_Device_Text := '';
L_Critical_Text := '';
L_Event_Text := '';
L_Add_Text := '';

// ======================================================
// SERVICE / OUT-OF-SERVICE FLAGS
// ======================================================
GVL_STATUS.G_Diagnostics.Backup_Pump_Out_Of_Service :=
    NOT GVL_CONFIG.G_Backup_Circulation_Pump_In_Service;

GVL_STATUS.G_Diagnostics.Electric_Heater_Out_Of_Service :=
    NOT GVL_CONFIG.G_Electric_Heater_In_Service;

IF GVL_STATUS.G_Diagnostics.Backup_Pump_Out_Of_Service THEN
    L_Any_Heating_Device_OOS := TRUE;
    L_Add_Text := 'backup pump out of service';
    L_Device_Text := L_Add_Text;
END_IF;

IF GVL_STATUS.G_Diagnostics.Electric_Heater_Out_Of_Service THEN
    L_Any_Heating_Device_OOS := TRUE;
    L_Add_Text := 'electric heater out of service';
    IF LEN(L_Device_Text) = 0 THEN
        L_Device_Text := L_Add_Text;
    ELSIF (LEN(L_Device_Text) + LEN(L_Add_Text) + 2) < 200 THEN
        L_Device_Text := CONCAT(L_Device_Text, CONCAT('; ', L_Add_Text));
    END_IF;
END_IF;

fbDiagEventManager(
    VI_Code := GVL_CONFIG.ERR_BACKUP_PUMP_OUT_OF_SERVICE,
    VI_Severity := 2,
    VI_Active := GVL_STATUS.G_Diagnostics.Backup_Pump_Out_Of_Service,
    VI_Timestamp := VI_System_Time_MS,
    VI_Source := 400,
    VIO_Events := GVL_STATUS.G_Diagnostics_Events,
    VIO_Count := GVL_STATUS.G_Diagnostics_Count
);

fbDiagEventManager(
    VI_Code := GVL_CONFIG.ERR_ELECTRIC_HEATER_OUT_OF_SERVICE,
    VI_Severity := 2,
    VI_Active := GVL_STATUS.G_Diagnostics.Electric_Heater_Out_Of_Service,
    VI_Timestamp := VI_System_Time_MS,
    VI_Source := 401,
    VIO_Events := GVL_STATUS.G_Diagnostics_Events,
    VIO_Count := GVL_STATUS.G_Diagnostics_Count
);

FOR L_i := 1 TO GVL_CONSTANTS.C_MAX_MANIFOLDS DO

    GVL_STATUS.G_Diagnostics.Manifold_Pump_Out_Of_Service[L_i] :=
        NOT GVL_CONFIG.G_Manifold_Pump_In_Service[L_i];

    IF GVL_STATUS.G_Diagnostics.Manifold_Pump_Out_Of_Service[L_i] THEN
        L_Any_Heating_Device_OOS := TRUE;
        L_Add_Text := CONCAT('manifold pump OOS #', INT_TO_STRING(L_i));

        IF LEN(L_Device_Text) = 0 THEN
            L_Device_Text := L_Add_Text;
        ELSIF (LEN(L_Device_Text) + LEN(L_Add_Text) + 2) < 200 THEN
            L_Device_Text := CONCAT(L_Device_Text, CONCAT('; ', L_Add_Text));
        END_IF;
    END_IF;

    fbDiagEventManager(
        VI_Code := GVL_CONFIG.ERR_MANIFOLD_PUMP_OUT_OF_SERVICE,
        VI_Severity := 2,
        VI_Active := GVL_STATUS.G_Diagnostics.Manifold_Pump_Out_Of_Service[L_i],
        VI_Timestamp := VI_System_Time_MS,
        VI_Source := 410 + L_i,
        VIO_Events := GVL_STATUS.G_Diagnostics_Events,
        VIO_Count := GVL_STATUS.G_Diagnostics_Count
    );

END_FOR;

GVL_STATUS.G_Diagnostics.DHW_Heating_Pump_Out_Of_Service :=
    NOT GVL_CONFIG.G_DHW_Heating_Pump_In_Service;

GVL_STATUS.G_Diagnostics.DHW_Circ_Pump_Out_Of_Service :=
    NOT GVL_CONFIG.G_DHW_Circ_Pump_In_Service;

IF GVL_STATUS.G_Diagnostics.DHW_Heating_Pump_Out_Of_Service THEN
    L_Any_Heating_Device_OOS := TRUE;
    L_Add_Text := 'DHW heating pump out of service';

    IF LEN(L_Device_Text) = 0 THEN
        L_Device_Text := L_Add_Text;
    ELSIF (LEN(L_Device_Text) + LEN(L_Add_Text) + 2) < 200 THEN
        L_Device_Text := CONCAT(L_Device_Text, CONCAT('; ', L_Add_Text));
    END_IF;
END_IF;

IF GVL_STATUS.G_Diagnostics.DHW_Circ_Pump_Out_Of_Service THEN
    L_Any_Heating_Device_OOS := TRUE;
    L_Add_Text := 'DHW circ pump out of service';

    IF LEN(L_Device_Text) = 0 THEN
        L_Device_Text := L_Add_Text;
    ELSIF (LEN(L_Device_Text) + LEN(L_Add_Text) + 2) < 200 THEN
        L_Device_Text := CONCAT(L_Device_Text, CONCAT('; ', L_Add_Text));
    END_IF;
END_IF;

fbDiagEventManager(
    VI_Code := GVL_CONFIG.ERR_DHW_HEATING_PUMP_OUT_OF_SERVICE,
    VI_Severity := 2,
    VI_Active := GVL_STATUS.G_Diagnostics.DHW_Heating_Pump_Out_Of_Service,
    VI_Timestamp := VI_System_Time_MS,
    VI_Source := 420,
    VIO_Events := GVL_STATUS.G_Diagnostics_Events,
    VIO_Count := GVL_STATUS.G_Diagnostics_Count
);

fbDiagEventManager(
    VI_Code := GVL_CONFIG.ERR_DHW_CIRC_PUMP_OUT_OF_SERVICE,
    VI_Severity := 2,
    VI_Active := GVL_STATUS.G_Diagnostics.DHW_Circ_Pump_Out_Of_Service,
    VI_Timestamp := VI_System_Time_MS,
    VI_Source := 421,
    VIO_Events := GVL_STATUS.G_Diagnostics_Events,
    VIO_Count := GVL_STATUS.G_Diagnostics_Count
);

// ======================================================
// FREEZE HARDWARE EVENT PROJECTION
// ======================================================
L_Critical_Fault := GVL_STATE.G_Freeze_Hardware_Failed;

IF L_Critical_Fault THEN
    L_Critical_Text := 'Freeze hardware critical fault';
END_IF;

fbDiagEventManager(
    VI_Code := GVL_CONFIG.ERR_FREEZE_HARDWARE_FAILED,
    VI_Severity := 4,
    VI_Active := L_Critical_Fault,
    VI_Timestamp := VI_System_Time_MS,
    VI_Source := 430,
    VIO_Events := GVL_STATUS.G_Diagnostics_Events,
    VIO_Count := GVL_STATUS.G_Diagnostics_Count
);

GVL_STATUS.G_Diagnostics.Freeze_Hardware_Event_Pending :=
    GVL_STATUS.G_Diagnostics.Freeze_Hardware_Event_Pending OR
    L_Critical_Fault OR
    L_Any_Heating_Device_OOS;

IF L_Critical_Fault AND L_Any_Heating_Device_OOS THEN
    L_Event_Text := CONCAT(L_Critical_Text, '; ');
    IF (LEN(L_Event_Text) + LEN(L_Device_Text)) < 200 THEN
        L_Event_Text := CONCAT(L_Event_Text, L_Device_Text);
    END_IF;
    GVL_STATUS.G_Diagnostics.Freeze_Hardware_Event_Text := L_Event_Text;
ELSIF L_Critical_Fault THEN
    GVL_STATUS.G_Diagnostics.Freeze_Hardware_Event_Text := L_Critical_Text;
ELSIF L_Any_Heating_Device_OOS THEN
    GVL_STATUS.G_Diagnostics.Freeze_Hardware_Event_Text := L_Device_Text;
END_IF;

VO_Executed := TRUE;
VO_Valid := TRUE;

END_FUNCTION_BLOCK
// >>> BULK_SYNC_ANCHOR: FB_Heating_Runtime_Diagnostics_Phase <<<

(* ---- FB_Heating_Runtime_Output_Projection_Phase.st ---- *)
// ==============================================================================
// Heating runtime output projection phase
// Final phase wrapper around physical output projection.
// Does NOT calculate heating logic and does NOT publish state/status.
// ==============================================================================
FUNCTION_BLOCK FB_Heating_Runtime_Output_Projection_Phase
VAR_INPUT
    VI_Enable : BOOL;
    VI_Zone_Valves : ARRAY[1..GVL_CONSTANTS.C_MAX_HEATING_CIRCUITS] OF BOOL;
    VI_Manifold_Pumps : ARRAY[1..GVL_CONSTANTS.C_MAX_MANIFOLDS] OF BOOL;
    VI_Manifold_Valves : ARRAY[1..GVL_CONSTANTS.C_MAX_MANIFOLDS] OF REAL;
    VI_DHW_Heating_Pump : BOOL;
    VI_DHW_Circ_Pump : BOOL;
    VI_Backup_Circulation_Pump : BOOL;
    VI_Electric_Heater_Enable : BOOL;
END_VAR
VAR_OUTPUT
    VO_Executed : BOOL;
    VO_Valid : BOOL;
END_VAR
VAR
    fbOutputProjection : FB_Heating_Output_Projection;
END_VAR

VO_Executed := FALSE;
VO_Valid := FALSE;

IF NOT VI_Enable THEN
    RETURN;
END_IF;

fbOutputProjection(
    VI_Zone_Valves := VI_Zone_Valves,
    VI_Manifold_Pumps := VI_Manifold_Pumps,
    VI_Manifold_Valves := VI_Manifold_Valves,
    VI_DHW_Heating_Pump := VI_DHW_Heating_Pump,
    VI_DHW_Circ_Pump := VI_DHW_Circ_Pump,
    VI_Backup_Circulation_Pump := VI_Backup_Circulation_Pump,
    VI_Electric_Heater_Enable := VI_Electric_Heater_Enable
);

VO_Executed := TRUE;
VO_Valid := TRUE;

END_FUNCTION_BLOCK
// >>> BULK_SYNC_ANCHOR: FB_Heating_Runtime_Output_Projection_Phase <<<

(* ---- FB_Heating_System_Manager.st ---- *)
FUNCTION_BLOCK FB_Heating_System_Manager
VAR_INPUT
    VI_System_Mode : E_System_Operating_Mode;
    VI_System_Time_MS : UDINT;
    VI_IsActivePLC : BOOL;
    VI_Outdoor_Temp : REAL;
    VI_Config : ST_Heating_Config;
    VI_Tariff : ST_Tariff_Config;
    VI_Current_Hour : UINT;
    VI_DHW_Heating_Demand : BOOL;
    VI_DHW_Target_Temp : REAL;
    VI_Emergency_Stop : BOOL;
    VI_Gas_Safety_Stop : BOOL;
    VI_Boiler_Error_Status : ARRAY[1..GVL_CONSTANTS.C_MAX_BOILERS] OF BOOL;
    VI_Boiler_OT_Online : ARRAY[1..GVL_CONSTANTS.C_MAX_BOILERS] OF BOOL;
    VI_Boiler_Modulation : ARRAY[1..GVL_CONSTANTS.C_MAX_BOILERS] OF REAL;
END_VAR
VAR_IN_OUT
    VI_Floor_Temps : ARRAY[1..GVL_CONSTANTS.C_MAX_HEATING_CIRCUITS] OF REAL;
    VI_Room_Temps : ARRAY[1..GVL_CONSTANTS.C_MAX_ZONES] OF REAL;
    VI_Manifold_Pressures : ARRAY[1..GVL_CONSTANTS.C_MAX_MANIFOLDS] OF REAL;
    VI_Manifold_Currents : ARRAY[1..GVL_CONSTANTS.C_MAX_MANIFOLDS] OF REAL;
    VI_Manifold_Temps_Supply : ARRAY[1..GVL_CONSTANTS.C_MAX_MANIFOLDS] OF REAL;
    VI_Manifold_Temps_Return : ARRAY[1..GVL_CONSTANTS.C_MAX_MANIFOLDS] OF REAL;
    VI_Boiler_Flame_Status : ARRAY[1..GVL_CONSTANTS.C_MAX_BOILERS] OF BOOL;
    VI_Zone_Configs : ARRAY[1..GVL_CONSTANTS.C_MAX_HEATING_CIRCUITS] OF ST_FloorHeating_Circuit_Config;
    VI_Rule_Actions : ARRAY[1..GVL_CONSTANTS.C_MAX_RULES] OF ST_Rule_Action;
    VI_IO_Modules_Online : ARRAY[1..GVL_CONSTANTS.C_MAX_MODULES] OF BOOL;
    VI_Manifold_End_Switches : ARRAY[1..GVL_CONSTANTS.C_MAX_MANIFOLDS] OF BOOL;
    VI_Valve_Test_Config : ARRAY[1..GVL_CONSTANTS.C_MAX_MANIFOLDS] OF ST_Valve_Test_Config;
END_VAR
VAR_OUTPUT
    VO_Manifold_Valves : ARRAY[1..GVL_CONSTANTS.C_MAX_MANIFOLDS] OF REAL;
    VO_Manifold_Pumps : ARRAY[1..GVL_CONSTANTS.C_MAX_MANIFOLDS] OF BOOL;
    VO_Zone_Valves : ARRAY[1..GVL_CONSTANTS.C_MAX_HEATING_CIRCUITS] OF BOOL;
    VO_Boiler_OT_Enable : ARRAY[1..GVL_CONSTANTS.C_MAX_BOILERS] OF BOOL;
    VO_Boiler_OT_Setpoint : ARRAY[1..GVL_CONSTANTS.C_MAX_BOILERS] OF REAL;
    VO_Backup_Circulation_Pump : BOOL;
    VO_Electric_Heater_Enable : BOOL;
    VO_Freeze_Risk_Status : BOOL;
    VO_Status : ARRAY[1..GVL_CONSTANTS.C_MAX_MANIFOLDS] OF ST_Manifold_Status;
    VO_Boiler_Status : ARRAY[1..GVL_CONSTANTS.C_MAX_BOILERS] OF ST_Boiler_Status;
END_VAR
VAR
    L_i : INT;
    L_Target_Supply_Temp : REAL;
    L_Manifold_Demand_Map : ARRAY[1..GVL_CONSTANTS.C_MAX_MANIFOLDS] OF BOOL;
    L_Manifold_Demand_Filtered : ARRAY[1..GVL_CONSTANTS.C_MAX_MANIFOLDS] OF BOOL;
    L_Manifold_Available : ARRAY[1..GVL_CONSTANTS.C_MAX_MANIFOLDS] OF BOOL;
    L_Manifold_In_Service : ARRAY[1..GVL_CONSTANTS.C_MAX_MANIFOLDS] OF BOOL;
    L_Manifold_Subsystem_Degraded : ARRAY[1..GVL_CONSTANTS.C_MAX_MANIFOLDS] OF BOOL;
    L_Manifold_Base_Priority : ARRAY[1..GVL_CONSTANTS.C_MAX_MANIFOLDS] OF INT;
    L_Manifold_Effective_Priority : ARRAY[1..GVL_CONSTANTS.C_MAX_MANIFOLDS] OF INT;
    L_Manifold_Thermal_Weight : ARRAY[1..GVL_CONSTANTS.C_MAX_MANIFOLDS] OF REAL;
    L_Allocation_Degraded : BOOL;
    fbValveTestManager : FB_Valve_Test_Manager;
    L_IO_Failsafe_Active : BOOL;
    L_Freeze_Active : BOOL;
    L_Freeze_Target_Supply : REAL;
    L_Policy_Degraded : BOOL;
    L_Sensor_Error : BOOL;
    L_Subsys_Degraded : BOOL;
    L_Pressure_OK : BOOL;
    L_Prev_Pressure : ARRAY[1..GVL_CONSTANTS.C_MAX_MANIFOLDS] OF REAL;
    L_Prev_Current : ARRAY[1..GVL_CONSTANTS.C_MAX_MANIFOLDS] OF REAL;
    L_Error_Instant : REAL;
    L_Confidence : REAL;
    L_Policy_Target_Adjustment : REAL;
    fbAdaptiveTarget : FB_Heating_Adaptive_Target;
    fbSafetyGate : FB_Heating_Safety_Gate;
    fbSafeState : FB_Heating_Safe_State;
    fbDemandMap : FB_Heating_Demand_Map;
    fbPolicyPriorityBridge : FB_Heating_Policy_Priority_Bridge;
    fbAllocationFilter : FB_Heating_Allocation_Filter;
    fbRuntimeObservability : FB_Heating_Runtime_Observability;
    fbCircuitControl : FB_Heating_Circuit_Control;
    fbManifoldControl : FB_Heating_Manifold_Control;
    fbBoilerControl : FB_Heating_Boiler_Control;
END_VAR

L_Policy_Degraded := (VI_System_Mode = E_System_Operating_Mode.MODE_DEGRADED);

GVL_STATE.G_Heating_IO_Fault := FALSE;
GVL_STATE.G_Heating_Sensor_Fault := FALSE;
GVL_STATE.G_Heating_Subsystem_Degraded := FALSE;
L_Sensor_Error := FALSE;
L_Subsys_Degraded := FALSE;
L_Allocation_Degraded := FALSE;

L_IO_Failsafe_Active := FALSE;
FOR L_i := 1 TO GVL_CONSTANTS.C_MAX_MODULES DO
    IF NOT VI_IO_Modules_Online[L_i] THEN
        L_IO_Failsafe_Active := TRUE;
        GVL_STATE.G_Heating_IO_Fault := TRUE;
        GVL_STATE.G_Heating_Subsystem_Degraded := TRUE;
        EXIT;
    END_IF;
END_FOR;

fbSafetyGate(
    VI_System_Mode := VI_System_Mode,
    VI_Emergency_Stop := VI_Emergency_Stop,
    VI_Gas_Safety_Stop := VI_Gas_Safety_Stop,
    VI_IO_Failsafe_Active := L_IO_Failsafe_Active,
    VI_Outdoor_Temp := VI_Outdoor_Temp,
    VI_Freeze_Threshold := VI_Config.Freeze_Threshold,
    VI_Floor_Temps := VI_Floor_Temps,
    VO_Freeze_Mode_Active => L_Freeze_Active,
    VO_Freeze_Target_Supply => L_Freeze_Target_Supply
);

fbSafeState(
    VI_Block_Normal_Heating := fbSafetyGate.VO_Block_Normal_Heating,
    VI_IO_Failsafe_Active := fbSafetyGate.VO_IO_Failsafe_Active,
    VI_Gas_Safety_Active := fbSafetyGate.VO_Gas_Safety_Active,
    VI_Freeze_Active := L_Freeze_Active,
    VI_Freeze_Target_Supply := L_Freeze_Target_Supply,
    VI_Manifold_Temps_Supply := VI_Manifold_Temps_Supply,
    VI_Boiler_Error_Status := VI_Boiler_Error_Status,
    VI_Boiler_OT_Online := VI_Boiler_OT_Online
);

IF fbSafeState.VO_Applied THEN
    FOR L_i := 1 TO GVL_CONSTANTS.C_MAX_HEATING_CIRCUITS DO
        VO_Zone_Valves[L_i] := fbSafeState.VO_Zone_Valves[L_i];
    END_FOR;

    FOR L_i := 1 TO GVL_CONSTANTS.C_MAX_MANIFOLDS DO
        VO_Manifold_Pumps[L_i] := fbSafeState.VO_Manifold_Pumps[L_i];
        VO_Manifold_Valves[L_i] := fbSafeState.VO_Manifold_Valves[L_i];
    END_FOR;

    FOR L_i := 1 TO GVL_CONSTANTS.C_MAX_BOILERS DO
        VO_Boiler_OT_Enable[L_i] := fbSafeState.VO_Boiler_OT_Enable[L_i];
        VO_Boiler_OT_Setpoint[L_i] := fbSafeState.VO_Boiler_OT_Setpoint[L_i];
        VO_Boiler_Status[L_i] := fbSafeState.VO_Boiler_Status[L_i];
    END_FOR;

    VO_Backup_Circulation_Pump := fbSafeState.VO_Backup_Circulation_Pump;
    VO_Electric_Heater_Enable := fbSafeState.VO_Electric_Heater_Enable;
    VO_Freeze_Risk_Status := fbSafeState.VO_Freeze_Risk_Status;
    RETURN;
END_IF;

VO_Backup_Circulation_Pump := FALSE;
VO_Electric_Heater_Enable := FALSE;
VO_Freeze_Risk_Status := FALSE;

IF L_Freeze_Active THEN
    L_Target_Supply_Temp := L_Freeze_Target_Supply;
ELSE
    L_Target_Supply_Temp := VI_Config.Target_Floor_Temp;
END_IF;

fbAdaptiveTarget(
    VI_Base_Target_Supply_Temp := L_Target_Supply_Temp,
    VI_Global_Target_Temperature := GVL_STATE.G_Target_Temperature,
    VI_Zone_Configs := VI_Zone_Configs,
    VI_Floor_Temps := VI_Floor_Temps,
    VI_Room_Temps := VI_Room_Temps,
    VO_Target_Supply_Temp => L_Target_Supply_Temp
);

L_Policy_Target_Adjustment := GVL_HEATING_POLICY.G_Policy_Target_Adjustment;

IF L_Policy_Target_Adjustment > REAL#5.0 THEN
    L_Policy_Target_Adjustment := REAL#5.0;
ELSIF L_Policy_Target_Adjustment < REAL#-3.0 THEN
    L_Policy_Target_Adjustment := REAL#-3.0;
END_IF;

L_Target_Supply_Temp :=
    LIMIT(
        GVL_CONSTANTS.C_BOILER_SETPOINT_MIN,
        L_Target_Supply_Temp + L_Policy_Target_Adjustment,
        GVL_CONSTANTS.C_BOILER_SETPOINT_MAX
    );

fbCircuitControl(
    VI_System_Time_MS := VI_System_Time_MS,
    VI_Current_Hour := VI_Current_Hour,
    VI_IsActivePLC := VI_IsActivePLC,
    VI_Config := VI_Config,
    VI_Tariff := VI_Tariff,
    VI_Scenario_Adjust := REAL#0.0,
    VI_Zone_Configs := VI_Zone_Configs,
    VI_Floor_Temps := VI_Floor_Temps,
    VI_Room_Temps := VI_Room_Temps,
    VI_Rule_Actions := VI_Rule_Actions,
    VO_Zone_Valves => VO_Zone_Valves,
    VO_Heating_Sensor_Fault => L_Sensor_Error
);

GVL_STATE.G_Heating_Sensor_Fault := L_Sensor_Error;

fbDemandMap(
    VI_Zone_Valves := VO_Zone_Valves,
    VI_Zone_Configs := VI_Zone_Configs,
    VO_Manifold_Demand_Map => L_Manifold_Demand_Map
);

FOR L_i := 1 TO GVL_CONSTANTS.C_MAX_MANIFOLDS DO
    L_Manifold_Available[L_i] := VI_Manifold_Pressures[L_i] >= GVL_CONSTANTS.C_MIN_HEATING_MANIFOLD_PRESSURE;
    L_Manifold_In_Service[L_i] := GVL_CONFIG.G_Manifold_Pump_In_Service[L_i];
    L_Manifold_Subsystem_Degraded[L_i] :=
        GVL_STATE.G_Predictive_Pump_Pressure_Drop[L_i]
        OR GVL_STATE.G_Predictive_Pump_Current_Rise[L_i];

    L_Manifold_Base_Priority[L_i] := GVL_CONFIG.G_Manifold_Priority[L_i];
    L_Manifold_Thermal_Weight[L_i] := GVL_CONFIG.G_Manifold_Thermal_Weight[L_i];
END_FOR;

fbPolicyPriorityBridge(
    VI_Enable := (GVL_CONFIG.G_Max_Thermal_Budget > REAL#0.0),
    VI_Zone_Valves := VO_Zone_Valves,
    VI_Zone_Configs := VI_Zone_Configs,
    VI_Manifold_Base_Priority := L_Manifold_Base_Priority,
    VI_Zone_Priority_Bias := GVL_HEATING_POLICY.G_Zone_Priority_Bias,
    VI_Policy_Priority_Multiplier := GVL_HEATING_POLICY.G_Policy_Priority_Multiplier,
    VO_Manifold_Effective_Priority => L_Manifold_Effective_Priority
);

fbAllocationFilter(
    VI_Enable := TRUE,
    VI_Enable_Policy_Allocation := (GVL_CONFIG.G_Max_Thermal_Budget > REAL#0.0),
    VI_Freeze_Mode_Active := L_Freeze_Active,
    VI_DHW_Heating_Demand := VI_DHW_Heating_Demand,
    VI_Manifold_Demand_Map := L_Manifold_Demand_Map,
    VI_Manifold_Available := L_Manifold_Available,
    VI_Manifold_In_Service := L_Manifold_In_Service,
    VI_Manifold_Subsystem_Degraded := L_Manifold_Subsystem_Degraded,
    VI_Manifold_Base_Priority := L_Manifold_Effective_Priority,
    VI_Manifold_Thermal_Weight := L_Manifold_Thermal_Weight,
    VI_Max_Thermal_Budget := GVL_CONFIG.G_Max_Thermal_Budget,
    VO_Manifold_Demand_Filtered => L_Manifold_Demand_Filtered,
    VO_Allocation_Degraded => L_Allocation_Degraded
);

fbRuntimeObservability(
    VI_Policy_Active := (GVL_CONFIG.G_Max_Thermal_Budget > REAL#0.0),
    VI_Freeze_Bypass_Active := L_Freeze_Active,
    VI_DHW_Bypass_Active := VI_DHW_Heating_Demand,
    VI_Budget_Max := GVL_CONFIG.G_Max_Thermal_Budget,
    VI_Budget_Used := fbAllocationFilter.VO_Thermal_Budget_Used,
    VI_Requested := L_Manifold_Demand_Map,
    VI_Allowed := fbAllocationFilter.VO_Manifold_Allowed,
    VI_Filtered := L_Manifold_Demand_Filtered,
    VI_Block_Reason := fbAllocationFilter.VO_Manifold_Block_Reason,
    VI_Effective_Priority := fbAllocationFilter.VO_Manifold_Priority_Effective,
    VI_Priority_Bridge_Active := fbPolicyPriorityBridge.VO_Bridge_Active,
    VI_Priority_Bias_Applied := fbPolicyPriorityBridge.VO_Manifold_Priority_Bias_Applied,
    VI_Priority_Effective := L_Manifold_Effective_Priority
);

IF L_Allocation_Degraded THEN
    GVL_STATE.G_Heating_Subsystem_Degraded := TRUE;
END_IF;

fbManifoldControl(
    VI_System_Time_MS := VI_System_Time_MS,
    VI_IsActivePLC := VI_IsActivePLC,
    VI_DHW_Heating_Demand := VI_DHW_Heating_Demand,
    VI_Freeze_Mode_Active := L_Freeze_Active,
    VI_Target_Supply_Temp := L_Target_Supply_Temp,
    VI_Any_Zone_Active := L_Manifold_Demand_Filtered,
    VI_Manifold_Pressures := VI_Manifold_Pressures,
    VI_Manifold_Currents := VI_Manifold_Currents,
    VI_Manifold_Temps_Supply := VI_Manifold_Temps_Supply,
    VI_Manifold_Temps_Return := VI_Manifold_Temps_Return,
    VO_Manifold_Pumps => VO_Manifold_Pumps,
    VO_Manifold_Valves => VO_Manifold_Valves,
    VO_Status => VO_Status
);

FOR L_i := 1 TO GVL_CONSTANTS.C_MAX_MANIFOLDS DO
    L_Pressure_OK := VI_Manifold_Pressures[L_i] >= GVL_CONSTANTS.C_MIN_HEATING_MANIFOLD_PRESSURE;

    IF VO_Manifold_Pumps[L_i] AND NOT L_Pressure_OK THEN
        VO_Manifold_Pumps[L_i] := FALSE;
        GVL_STATE.G_Heating_Subsystem_Degraded := TRUE;
    END_IF;

    IF (L_Prev_Pressure[L_i] > REAL#0.0) AND ((L_Prev_Pressure[L_i] - VI_Manifold_Pressures[L_i]) > REAL#0.2) THEN
        GVL_STATE.G_Predictive_Pump_Pressure_Drop[L_i] := TRUE;
    ELSE
        GVL_STATE.G_Predictive_Pump_Pressure_Drop[L_i] := FALSE;
    END_IF;

    IF (L_Prev_Current[L_i] > REAL#0.0) AND (VI_Manifold_Currents[L_i] > (L_Prev_Current[L_i] * REAL#1.2)) THEN
        GVL_STATE.G_Predictive_Pump_Current_Rise[L_i] := TRUE;
    ELSE
        GVL_STATE.G_Predictive_Pump_Current_Rise[L_i] := FALSE;
    END_IF;

    IF GVL_STATE.G_Predictive_Pump_Pressure_Drop[L_i] OR GVL_STATE.G_Predictive_Pump_Current_Rise[L_i] THEN
        GVL_STATE.G_Heating_Subsystem_Degraded := TRUE;
    END_IF;

    L_Prev_Pressure[L_i] := VI_Manifold_Pressures[L_i];
    L_Prev_Current[L_i] := VI_Manifold_Currents[L_i];
END_FOR;

L_Error_Instant := REAL#0.0;

IF GVL_STATE.G_Heating_Sensor_Fault THEN
    L_Error_Instant := L_Error_Instant + REAL#0.2;
END_IF;

IF GVL_STATE.G_Heating_IO_Fault THEN
    L_Error_Instant := L_Error_Instant + REAL#0.2;
END_IF;

FOR L_i := 1 TO GVL_CONSTANTS.C_MAX_MANIFOLDS DO
    IF VI_Manifold_Pressures[L_i] < GVL_CONSTANTS.C_MIN_HEATING_MANIFOLD_PRESSURE THEN
        L_Error_Instant := L_Error_Instant + REAL#0.1;
        EXIT;
    END_IF;
END_FOR;

FOR L_i := 1 TO GVL_CONSTANTS.C_MAX_MANIFOLDS DO
    IF GVL_STATE.G_Predictive_Pump_Pressure_Drop[L_i] OR GVL_STATE.G_Predictive_Pump_Current_Rise[L_i] THEN
        L_Error_Instant := L_Error_Instant + REAL#0.2;
        EXIT;
    END_IF;
END_FOR;

GVL_STATE.G_Heating_Error_Score := (GVL_STATE.G_Heating_Error_Score * REAL#0.98) + L_Error_Instant;
L_Confidence := REAL#1.0 - GVL_STATE.G_Heating_Error_Score;

IF L_Confidence < REAL#0.0 THEN
    L_Confidence := REAL#0.0;
ELSIF L_Confidence > REAL#1.0 THEN
    L_Confidence := REAL#1.0;
END_IF;

GVL_STATE.G_Heating_Confidence := L_Confidence;

GVL_STATE.G_Heating_Confidence_Reason_Code := 0;
GVL_STATE.G_Heating_Confidence_Reason_Text := 'OK';

IF GVL_STATE.G_Heating_IO_Fault THEN
    GVL_STATE.G_Heating_Confidence_Reason_Code := 2;
    GVL_STATE.G_Heating_Confidence_Reason_Text := 'IO fault detected';
ELSIF GVL_STATE.G_Heating_Sensor_Fault THEN
    GVL_STATE.G_Heating_Confidence_Reason_Code := 1;
    GVL_STATE.G_Heating_Confidence_Reason_Text := 'Sensor fault detected';
ELSE
    FOR L_i := 1 TO GVL_CONSTANTS.C_MAX_MANIFOLDS DO
        IF VI_Manifold_Pressures[L_i] < GVL_CONSTANTS.C_MIN_HEATING_MANIFOLD_PRESSURE THEN
            GVL_STATE.G_Heating_Confidence_Reason_Code := 3;
            GVL_STATE.G_Heating_Confidence_Reason_Text := 'Low manifold pressure';
            EXIT;
        END_IF;
    END_FOR;

    FOR L_i := 1 TO GVL_CONSTANTS.C_MAX_MANIFOLDS DO
        IF GVL_STATE.G_Predictive_Pump_Pressure_Drop[L_i] OR GVL_STATE.G_Predictive_Pump_Current_Rise[L_i] THEN
            GVL_STATE.G_Heating_Confidence_Reason_Code := 4;
            GVL_STATE.G_Heating_Confidence_Reason_Text := 'Predictive pump degradation';
            EXIT;
        END_IF;
    END_FOR;
END_IF;

IF GVL_STATE.G_Heating_Confidence < REAL#0.5 THEN
    L_Target_Supply_Temp := L_Target_Supply_Temp - REAL#3.0;
END_IF;

CASE GVL_STATE.G_Heating_Confidence_Reason_Code OF
    1:
        L_Target_Supply_Temp := LIMIT(GVL_CONSTANTS.C_BOILER_SETPOINT_MIN, REAL#40.0, GVL_CONSTANTS.C_BOILER_SETPOINT_MAX);
    2:
        VO_Backup_Circulation_Pump := TRUE;
    3:
        FOR L_i := 1 TO GVL_CONSTANTS.C_MAX_MANIFOLDS DO
            VO_Manifold_Pumps[L_i] := FALSE;
        END_FOR;
    4:
        L_Target_Supply_Temp := LIMIT(GVL_CONSTANTS.C_BOILER_SETPOINT_MIN, L_Target_Supply_Temp - REAL#5.0, GVL_CONSTANTS.C_BOILER_SETPOINT_MAX);
ELSE
    // no auto-recovery action
END_CASE;

fbValveTestManager(
    VI_System_Time_MS := VI_System_Time_MS,
    VI_IsActivePLC := VI_IsActivePLC,
    VI_Valve_Currents := VI_Manifold_Currents,
    VI_Valve_End_Switches := VI_Manifold_End_Switches,
    VI_Config := VI_Valve_Test_Config
);

IF fbValveTestManager.VO_Test_Active THEN
    L_i := fbValveTestManager.VO_Current_Valve;
    IF L_i >= 1 AND L_i <= GVL_CONSTANTS.C_MAX_MANIFOLDS THEN
        IF fbValveTestManager.VO_Valve_Cmd[L_i] THEN
            VO_Manifold_Valves[L_i] := REAL#100.0;
        ELSE
            VO_Manifold_Valves[L_i] := REAL#0.0;
        END_IF;
        VO_Manifold_Pumps[L_i] := FALSE;
    END_IF;
END_IF;

fbBoilerControl(
    VI_System_Time_MS := VI_System_Time_MS,
    VI_IsActivePLC := VI_IsActivePLC,
    VI_DHW_Heating_Demand := VI_DHW_Heating_Demand,
    VI_DHW_Target_Temp := VI_DHW_Target_Temp,
    VI_Target_Supply_Temp := L_Target_Supply_Temp,
    VI_Freeze_Mode_Active := L_Freeze_Active,
    VI_Policy_Degraded := L_Policy_Degraded,
    VI_Manifold_Pumps := VO_Manifold_Pumps,
    VI_Manifold_Valves := VO_Manifold_Valves,
    VI_Boiler_Flame_Status := VI_Boiler_Flame_Status,
    VI_Boiler_Error_Status := VI_Boiler_Error_Status,
    VI_Boiler_OT_Online := VI_Boiler_OT_Online,
    VI_Boiler_Modulation := VI_Boiler_Modulation,
    VO_Boiler_OT_Enable => VO_Boiler_OT_Enable,
    VO_Boiler_OT_Setpoint => VO_Boiler_OT_Setpoint,
    VO_Boiler_Status => VO_Boiler_Status,
    VO_Any_Subsystem_Degraded => L_Subsys_Degraded
);

GVL_STATE.G_Heating_Subsystem_Degraded := GVL_STATE.G_Heating_Subsystem_Degraded OR L_Subsys_Degraded;

END_FUNCTION_BLOCK
// >>> BULK_SYNC_ANCHOR: FB_Heating_System_Manager <<<

(* ---- FB_Heating_Thermal_Model.st ---- *)
FUNCTION_BLOCK FB_Heating_Thermal_Model
VAR
    L_i : INT;
    L_DeltaT : REAL;
    L_Loss : REAL;
    L_Gain : REAL;
    L_Outdoor : REAL;
END_VAR

L_Outdoor := GVL_STATE.G_Outdoor_Temp;

FOR L_i := 1 TO GVL_CONSTANTS.C_MAX_ZONES DO

    L_DeltaT := GVL_STATE.G_Room_Temps[L_i] - L_Outdoor;

    L_Loss := L_DeltaT * REAL#0.01 * GVL_HEATING_POLICY.G_Zone_Thermal_Inertia[L_i];

    L_Gain := (GVL_STATE.G_Floor_Temps[L_i] - GVL_STATE.G_Room_Temps[L_i]) * REAL#0.05;

    GVL_HEATING_POLICY.G_Zone_Heat_Loss_Rate[L_i] := L_Loss;
    GVL_HEATING_POLICY.G_Zone_Heat_Gain_Rate[L_i] := L_Gain;

    GVL_HEATING_POLICY.G_Zone_Thermal_Response[L_i] := L_Gain - L_Loss;

    GVL_HEATING_POLICY.G_Zone_Thermal_Demand[L_i] :=
        GVL_STATE.G_Target_Temperature - GVL_STATE.G_Room_Temps[L_i];

    IF ABS(GVL_HEATING_POLICY.G_Zone_Thermal_Response[L_i]) > REAL#0.01 THEN
        GVL_HEATING_POLICY.G_Zone_Time_To_Heat_MS[L_i] :=
            REAL_TO_UDINT(ABS(GVL_HEATING_POLICY.G_Zone_Thermal_Demand[L_i] /
                  GVL_HEATING_POLICY.G_Zone_Thermal_Response[L_i]) * REAL#60000.0);
    ELSE
        GVL_HEATING_POLICY.G_Zone_Time_To_Heat_MS[L_i] := 0;
    END_IF;

    GVL_HEATING_POLICY.G_Zone_Predicted_Temp_30m[L_i] :=
        GVL_STATE.G_Room_Temps[L_i] +
        GVL_HEATING_POLICY.G_Zone_Thermal_Response[L_i] * REAL#30.0;

    GVL_HEATING_POLICY.G_Zone_Thermal_Model_Confidence[L_i] :=
        LIMIT(REAL#0.0, REAL#1.0, ABS(GVL_HEATING_POLICY.G_Zone_Thermal_Response[L_i]));

END_FOR;

END_FUNCTION_BLOCK

(* ---- FB_Modbus_RTU_TX_Builder.st ---- *)
FUNCTION_BLOCK FB_Modbus_RTU_TX_Builder
VAR_INPUT
    VI_Request_Valid : BOOL;
    VI_Slave_ID : BYTE;
    VI_Function_Code : E_Modbus_Function;
    VI_Start_Register : UINT;
    VI_Register_Count : UINT;
    VI_Write_Value : ARRAY[1..32] OF WORD;
END_VAR

VAR_OUTPUT
    VO_Frame : ST_Modbus_RTU_Frame;
    VO_Error : BOOL;
    VO_Error_Code : WORD;
END_VAR

VAR
    L_i : INT;
    L_j : INT;
    L_Pos : UINT;
    L_CRC : WORD;
    L_Byte_Count : UINT;
    L_Function_Byte : BYTE;
END_VAR

// ======================================================
// MODBUS RTU TX FRAME BUILDER
// ======================================================
// Builds Modbus RTU request frames only.
// This FB does not send data and does not modify response state.
// ======================================================

VO_Error := FALSE;
VO_Error_Code := 0;
VO_Frame.Valid := FALSE;
VO_Frame.Length := 0;
VO_Frame.CRC := 0;
L_Function_Byte := 0;

FOR L_i := 0 TO 255 DO
    VO_Frame.Data[L_i] := 0;
END_FOR;

IF NOT VI_Request_Valid THEN
    RETURN;
END_IF;

IF VI_Slave_ID = 0 THEN
    VO_Error := TRUE;
    VO_Error_Code := 16#0101;
    RETURN;
END_IF;

IF (VI_Register_Count = 0) OR (VI_Register_Count > 32) THEN
    VO_Error := TRUE;
    VO_Error_Code := 16#0102;
    RETURN;
END_IF;

CASE VI_Function_Code OF
    MB_FC03_READ_HOLDING_REGISTERS:
        L_Function_Byte := 3;
    MB_FC04_READ_INPUT_REGISTERS:
        L_Function_Byte := 4;
    MB_FC06_WRITE_SINGLE_REGISTER:
        L_Function_Byte := 6;
    MB_FC16_WRITE_MULTIPLE_REGISTERS:
        L_Function_Byte := 16;
ELSE
    VO_Error := TRUE;
    VO_Error_Code := 16#0104;
    RETURN;
END_CASE;

VO_Frame.Data[0] := VI_Slave_ID;
VO_Frame.Data[1] := L_Function_Byte;
VO_Frame.Data[2] := WORD_TO_BYTE(SHR(UINT_TO_WORD(VI_Start_Register), 8));
VO_Frame.Data[3] := WORD_TO_BYTE(UINT_TO_WORD(VI_Start_Register) AND 16#00FF);

CASE VI_Function_Code OF

    MB_FC03_READ_HOLDING_REGISTERS,
    MB_FC04_READ_INPUT_REGISTERS:

        VO_Frame.Data[4] := WORD_TO_BYTE(SHR(UINT_TO_WORD(VI_Register_Count), 8));
        VO_Frame.Data[5] := WORD_TO_BYTE(UINT_TO_WORD(VI_Register_Count) AND 16#00FF);
        VO_Frame.Length := 6;

    MB_FC06_WRITE_SINGLE_REGISTER:

        VO_Frame.Data[4] := WORD_TO_BYTE(SHR(VI_Write_Value[1], 8));
        VO_Frame.Data[5] := WORD_TO_BYTE(VI_Write_Value[1] AND 16#00FF);
        VO_Frame.Length := 6;

    MB_FC16_WRITE_MULTIPLE_REGISTERS:

        L_Byte_Count := VI_Register_Count * 2;

        IF L_Byte_Count > 64 THEN
            VO_Error := TRUE;
            VO_Error_Code := 16#0103;
            RETURN;
        END_IF;

        VO_Frame.Data[4] := WORD_TO_BYTE(SHR(UINT_TO_WORD(VI_Register_Count), 8));
        VO_Frame.Data[5] := WORD_TO_BYTE(UINT_TO_WORD(VI_Register_Count) AND 16#00FF);
        VO_Frame.Data[6] := UINT_TO_BYTE(L_Byte_Count);

        L_Pos := 7;

        FOR L_i := 1 TO UINT_TO_INT(VI_Register_Count) DO
            VO_Frame.Data[L_Pos] := WORD_TO_BYTE(SHR(VI_Write_Value[L_i], 8));
            VO_Frame.Data[L_Pos + 1] := WORD_TO_BYTE(VI_Write_Value[L_i] AND 16#00FF);
            L_Pos := L_Pos + 2;
        END_FOR;

        VO_Frame.Length := 7 + L_Byte_Count;

ELSE
    VO_Error := TRUE;
    VO_Error_Code := 16#0104;
    RETURN;
END_CASE;

// ======================================================
// INLINE MODBUS RTU CRC16
// ======================================================
L_CRC := 16#FFFF;

FOR L_i := 0 TO (UINT_TO_INT(VO_Frame.Length) - 1) DO

    L_CRC := L_CRC XOR BYTE_TO_WORD(VO_Frame.Data[L_i]);

    FOR L_j := 0 TO 7 DO
        IF (L_CRC AND 16#0001) <> 0 THEN
            L_CRC := SHR(L_CRC, 1);
            L_CRC := L_CRC XOR 16#A001;
        ELSE
            L_CRC := SHR(L_CRC, 1);
        END_IF;
    END_FOR;

END_FOR;

VO_Frame.CRC := L_CRC;
VO_Frame.Data[VO_Frame.Length] := WORD_TO_BYTE(L_CRC AND 16#00FF);
VO_Frame.Data[VO_Frame.Length + 1] := WORD_TO_BYTE(SHR(L_CRC, 8));
VO_Frame.Length := VO_Frame.Length + 2;
VO_Frame.Valid := TRUE;

END_FUNCTION_BLOCK

(* ---- FB_Mode_Manager.st ---- *)
FUNCTION_BLOCK FB_Mode_Manager

VAR_INPUT
    VI_Is_Night : BOOL;
    VI_Away_Request : BOOL;
    VI_Maintenance_Request : BOOL;
    VI_System_Time_MS : UDINT;
END_VAR

VAR_OUTPUT
    VO_Mode : E_Behavior_Mode;
    VO_Mode_Code : UDINT;
END_VAR

// default
VO_Mode := BEHAVIOR_HOME;
VO_Mode_Code := 0;

// priority-based transitions
IF VI_Maintenance_Request THEN
    VO_Mode := BEHAVIOR_MAINTENANCE;
    VO_Mode_Code := 300;
ELSIF VI_Away_Request THEN
    VO_Mode := BEHAVIOR_AWAY;
    VO_Mode_Code := 200;
ELSIF VI_Is_Night THEN
    VO_Mode := BEHAVIOR_NIGHT;
    VO_Mode_Code := 100;
END_IF;
END_FUNCTION_BLOCK

(* ---- FB_Scenario_Manager.st ---- *)
FUNCTION_BLOCK FB_Scenario_Manager
VAR_INPUT
    VI_Preheat_Request : BOOL;
    VI_System_Time_MS : UDINT; // Системное время (мс)
    VI_Activate_Request : E_SCENARIO_TYPE; // Запрос на активацию сценария
    VI_IsActivePLC : BOOL; // Флаг: Данный ПЛК является ведущим
    VI_System_Mode : E_System_Operating_Mode; // Агрегированный режим работы системы
END_VAR
VAR_OUTPUT
    VO_Current_Scenario : E_SCENARIO_TYPE; // Текущий активный сценарий
    VO_Status_Msg : STRING(200); // Строковое сообщение о статусе
END_VAR

VAR
    L_Last_Scenario_Time : UDINT;
    L_Requested_Scenario : E_SCENARIO_TYPE;
END_VAR

IF NOT VI_IsActivePLC THEN
    RETURN;
END_IF;

L_Requested_Scenario := VI_Activate_Request;

CASE VI_System_Mode OF
    E_System_Operating_Mode.MODE_SAFE_STOP,
    E_System_Operating_Mode.MODE_FREEZE_PROTECTION:
        IF VO_Current_Scenario <> E_SCENARIO_TYPE.SCENARIO_NONE THEN
            VO_Current_Scenario := E_SCENARIO_TYPE.SCENARIO_NONE;
            VO_Status_Msg := 'Сценарии принудительно отключены режимом безопасности';
        END_IF;
        RETURN;

    E_System_Operating_Mode.MODE_DEGRADED:
        CASE L_Requested_Scenario OF
            E_SCENARIO_TYPE.SCENARIO_NONE,
            E_SCENARIO_TYPE.SCENARIO_AWAY,
            E_SCENARIO_TYPE.SCENARIO_SLEEP,
            E_SCENARIO_TYPE.SCENARIO_PRESENCE:
                VO_Status_Msg := 'Сценарии работают в ограниченном degraded-режиме';
        ELSE
                L_Requested_Scenario := E_SCENARIO_TYPE.SCENARIO_NONE;
                VO_Status_Msg := 'Небезопасный сценарий заблокирован degraded-режимом';
        END_CASE;
ELSE
        // Normal mode: no additional clamp required.
END_CASE;

IF L_Requested_Scenario <> VO_Current_Scenario THEN
    // Проверка минимального времени работы сценария
    IF (VI_System_Time_MS - L_Last_Scenario_Time) >= 60000 OR VO_Current_Scenario = E_SCENARIO_TYPE.SCENARIO_NONE THEN
        // Логика переключения сценариев
        VO_Current_Scenario := L_Requested_Scenario;
        L_Last_Scenario_Time := VI_System_Time_MS;

        CASE VO_Current_Scenario OF
        E_SCENARIO_TYPE.SCENARIO_NONE:
            VO_Status_Msg := 'Сценарии отключены';
        E_SCENARIO_TYPE.SCENARIO_AWAY:
            VO_Status_Msg := 'Активирован сценарий: Вне дома (Охрана + Энергосбережение)';
        E_SCENARIO_TYPE.SCENARIO_SLEEP:
            VO_Status_Msg := 'Активирован сценарий: Сон (Ночное освещение + Климат)';
        E_SCENARIO_TYPE.SCENARIO_PRESENCE:
            VO_Status_Msg := 'Активирован сценарий: Имитация присутствия';
        ELSE
            VO_Status_Msg := 'Активирован сценарий';
        END_CASE;
    END_IF;
END_IF;

// --- PREHEAT SCENARIO INSERT ---
IF VI_Preheat_Request THEN
    // removed: direct heating write (moved to Heating Manager)
END_IF;

// >>> BULK_SYNC_ANCHOR: FB_Scenario_Manager <<<
END_FUNCTION_BLOCK

(* ---- FB_Simulation_Manager.st ---- *)
FUNCTION_BLOCK FB_Simulation_Manager
VAR_INPUT
    VI_System_Time_MS : UDINT;
    VI_IsActivePLC    : BOOL;
    VI_Scenario       : E_SCENARIO_TYPE;
    VI_Config         : ST_Scenario_Config;
END_VAR
VAR_OUTPUT
    VO_Sim_Lights     : ARRAY[1..32] OF BOOL;
    VO_Sim_Active     : BOOL;
    VO_Sim_Water_Leak : ARRAY[1..GVL_CONSTANTS.C_MAX_FLOOD_SENSORS] OF BOOL;
    VO_Sim_Gas_Leak   : ARRAY[1..GVL_CONSTANTS.C_MAX_METHANE_SENSORS] OF REAL;
END_VAR
VAR
    L_Last_Toggle     : UDINT;
    L_i               : INT;
    L_Slot            : UDINT;
END_VAR

IF (NOT VI_IsActivePLC) THEN
    VO_Sim_Active := FALSE;
    FOR L_i := 1 TO 32 DO
        VO_Sim_Lights[L_i] := FALSE;
    END_FOR;
    FOR L_i := 1 TO GVL_CONSTANTS.C_MAX_FLOOD_SENSORS DO
        VO_Sim_Water_Leak[L_i] := FALSE;
    END_FOR;
    FOR L_i := 1 TO GVL_CONSTANTS.C_MAX_METHANE_SENSORS DO
        VO_Sim_Gas_Leak[L_i] := REAL#0.0;
    END_FOR;
    RETURN;
END_IF;

IF (VI_Scenario = E_SCENARIO_TYPE.SCENARIO_AWAY) AND VI_Config.Presence_Simulation_Enabled THEN
    VO_Sim_Active := TRUE;

    IF (VI_System_Time_MS - L_Last_Toggle) >= (GVL_CONSTANTS.C_MS_IN_MINUTE * 30) THEN
        L_Last_Toggle := VI_System_Time_MS;
        L_Slot := (VI_System_Time_MS / GVL_CONSTANTS.C_MS_IN_MINUTE) MOD 32;

        FOR L_i := 1 TO 32 DO
            VO_Sim_Lights[L_i] := ((TO_UDINT(L_i) + L_Slot) MOD 5) = 0;
        END_FOR;
    END_IF;
ELSE
    VO_Sim_Active := FALSE;
    FOR L_i := 1 TO 32 DO
        VO_Sim_Lights[L_i] := FALSE;
    END_FOR;
END_IF;

FOR L_i := 1 TO GVL_CONSTANTS.C_MAX_FLOOD_SENSORS DO
    VO_Sim_Water_Leak[L_i] := FALSE;
END_FOR;
FOR L_i := 1 TO GVL_CONSTANTS.C_MAX_METHANE_SENSORS DO
    VO_Sim_Gas_Leak[L_i] := REAL#0.0;
END_FOR;

// >>> BULK_SYNC_ANCHOR: FB_Simulation_Manager <<<
END_FUNCTION_BLOCK

(* ---- FB_State_Manager.st ---- *)
FUNCTION_BLOCK FB_State_Manager
VAR_INPUT
    VI_System_Severity : E_System_Severity;
    VI_Root_Cause      : E_System_Root_Cause;
    VI_Freeze_Risk     : BOOL := FALSE;
END_VAR

VAR_OUTPUT
    VO_System_OK        : BOOL;
    VO_System_Warning   : BOOL;
    VO_System_Critical  : BOOL;
    VO_Status_Msg       : STRING(200);

    // compatibility output for existing orchestration
    VO_System_Mode      : E_System_Operating_Mode;
END_VAR

VO_System_OK := FALSE;
VO_System_Warning := FALSE;
VO_System_Critical := FALSE;
VO_Status_Msg := '';
VO_System_Mode := E_System_Operating_Mode.MODE_NORMAL;

CASE VI_System_Severity OF
    E_System_Severity.SEV_NORMAL:
        VO_System_OK := TRUE;
        VO_Status_Msg := 'Система в норме';
        VO_System_Mode := E_System_Operating_Mode.MODE_NORMAL;

    E_System_Severity.SEV_WARNING:
        VO_System_Warning := TRUE;
        VO_System_Mode := E_System_Operating_Mode.MODE_DEGRADED;
        CASE VI_Root_Cause OF
            E_System_Root_Cause.ROOT_WATER_LEAK:
                VO_Status_Msg := 'Предупреждение: протечка воды';
            E_System_Root_Cause.ROOT_CO_WARNING:
                VO_Status_Msg := 'Предупреждение: повышенный CO';
            ELSE
                VO_Status_Msg := 'Предупреждение системы';
        END_CASE;

    E_System_Severity.SEV_DEGRADED:
        VO_System_Warning := TRUE;
        VO_System_Mode := E_System_Operating_Mode.MODE_DEGRADED;
        CASE VI_Root_Cause OF
            E_System_Root_Cause.ROOT_SENSOR_FAULT:
                VO_Status_Msg := 'Деградация: ошибка датчика';
            E_System_Root_Cause.ROOT_IO_OFFLINE:
                VO_Status_Msg := 'Деградация: модуль IO недоступен';
            E_System_Root_Cause.ROOT_COMM_FAULT:
                VO_Status_Msg := 'Деградация: ошибка связи';
            E_System_Root_Cause.ROOT_WATCHDOG_FAULT:
                VO_Status_Msg := 'Деградация: watchdog fault';
            E_System_Root_Cause.ROOT_SUBSYSTEM_FAULT:
                VO_Status_Msg := 'Деградация: ошибка подсистемы';
            ELSE
                VO_Status_Msg := 'Деградация системы';
        END_CASE;

    E_System_Severity.SEV_CRITICAL:
        VO_System_Critical := TRUE;

        IF (VI_Root_Cause = E_System_Root_Cause.ROOT_GAS_LEAK OR
            VI_Root_Cause = E_System_Root_Cause.ROOT_CO_CRITICAL) AND
            VI_Freeze_Risk THEN
            VO_System_Mode := E_System_Operating_Mode.MODE_FREEZE_PROTECTION;
        ELSE
            VO_System_Mode := E_System_Operating_Mode.MODE_SAFE_STOP;
        END_IF;

        CASE VI_Root_Cause OF
            E_System_Root_Cause.ROOT_FIRE:
                VO_Status_Msg := 'АВАРИЯ: ПОЖАР';
            E_System_Root_Cause.ROOT_GAS_LEAK:
                VO_Status_Msg := 'АВАРИЯ: УТЕЧКА ГАЗА';
            E_System_Root_Cause.ROOT_CO_CRITICAL:
                VO_Status_Msg := 'АВАРИЯ: КРИТИЧЕСКИЙ CO';
            E_System_Root_Cause.ROOT_WATCHDOG_FAULT:
                VO_Status_Msg := 'АВАРИЯ: WATCHDOG';
            ELSE
                VO_Status_Msg := 'АВАРИЯ СИСТЕМЫ';
        END_CASE;
END_CASE;
// >>> BULK_SYNC_ANCHOR: FB_State_Manager <<<
END_FUNCTION_BLOCK

(* ---- FB_System_Health_Orchestrator.st ---- *)
// ==============================================================================
// System health orchestrator helper
//
// Internal helper for PRG_System.
// Owns safety latch update, watchdog, system health aggregation,
// system mode calculation, HMI/fault publication, diagnostic exports,
// and human-readable mode/cause text projection.
// ==============================================================================
FUNCTION_BLOCK FB_System_Health_Orchestrator
VAR_OUTPUT
    VO_First_Fault_Active : BOOL;
    VO_First_Fault_Type : INT;
    VO_First_Fault_Source : INT;
    VO_System_Severity : E_System_Severity;
    VO_Root_Cause : E_System_Root_Cause;
    VO_Watchdog_Fault : BOOL;
END_VAR

VAR
    fbSafety : FB_Safety_Manager;
    fbWatchdog : FB_Watchdog;
    fbSystemHealth : FB_System_Health;
    fbStateManager : FB_State_Manager;
    fbHMIInterface : FB_HMI_Interface;
    fbFaultLogger : FB_Fault_Logger;
END_VAR

fbSafety(
    VI_Gas_Alarm := GVL_STATE.G_Safety_Gas_Alarm,
    VI_Leak_Alarm := GVL_STATE.G_Safety_Leak_Alarm,
    VI_Smoke_Alarm := GVL_STATE.G_Safety_Smoke_Alarm,
    VI_Reset := GVL_COMMAND.G_Reset_Errors,
    VO_Gas_Latched => GVL_STATE.G_Safety_Gas_Latched,
    VO_Leak_Latched => GVL_STATE.G_Safety_Leak_Latched,
    VO_Smoke_Latched => GVL_STATE.G_Safety_Smoke_Latched,
    VO_Emergency_Stop => GVL_STATE.G_Safety_Emergency_Stop
);

GVL_STATE.G_Freeze_Hardware_Degraded := GVL_STATUS.G_Diagnostics.Backup_Pump_Fault OR GVL_STATUS.G_Diagnostics.Electric_Heater_Fault;
GVL_STATE.G_Freeze_Hardware_Failed := GVL_STATUS.G_Diagnostics.Backup_Pump_Fault AND GVL_STATUS.G_Diagnostics.Electric_Heater_Fault;

fbWatchdog(
    VI_System_Time_MS := GVL_STATUS.G_System_Time_MS
);

fbSystemHealth(
    VI_Smoke_Detected := GVL_HEALTH_BRIDGE.G_Smoke_Detected OR GVL_STATE.G_Safety_Smoke_Latched,
    VI_Gas_Detected := GVL_HEALTH_BRIDGE.G_Gas_Detected OR GVL_STATE.G_Safety_Gas_Latched,
    VI_CO_Warning_Level := GVL_HEALTH_BRIDGE.G_CO_Warning_Level,
    VI_CO_Alarm_Level := GVL_HEALTH_BRIDGE.G_CO_Alarm_Level,
    VI_Leak_Detected := GVL_HEALTH_BRIDGE.G_Leak_Detected OR GVL_STATE.G_Safety_Leak_Latched,
    VI_Sensor_Fault := GVL_STATE.G_Heating_Sensor_Fault OR GVL_STATE.G_DHW_Sensor_Fault OR GVL_STATUS.G_Diagnostics.Manifold_Pressure_Fault_Active OR GVL_STATUS.G_Diagnostics.Manifold_Current_Fault_Active OR GVL_STATUS.G_Diagnostics.Manifold_Return_Temp_Fault_Active,
    VI_IO_Offline := GVL_STATE.G_Heating_IO_Fault OR GVL_STATE.G_DHW_IO_Fault OR GVL_STATE.G_Ventilation_IO_Fault OR GVL_STATE.G_Lighting_IO_Fault,
    VI_Comm_Fault := GVL_STATE.G_Access_Comm_Fault,
    VI_Watchdog_Fault := fbWatchdog.VO_Watchdog_Fault,
    VI_Subsystem_Fault := GVL_STATE.G_Heating_Subsystem_Degraded OR GVL_STATE.G_DHW_Subsystem_Degraded OR GVL_STATE.G_Ventilation_Subsystem_Degraded OR GVL_STATUS.G_Diagnostics.Manifold_Pressure_Fault_Active OR GVL_STATUS.G_Diagnostics.Manifold_Current_Fault_Active OR GVL_STATUS.G_Diagnostics.Manifold_Return_Temp_Fault_Active
);

fbStateManager(
    VI_System_Severity := fbSystemHealth.VO_System_Severity,
    VI_Root_Cause := fbSystemHealth.VO_Root_Cause,
    VI_Freeze_Risk := GVL_STATE.G_Safety_Freeze_Risk
);

fbHMIInterface(
    VI_Severity := fbSystemHealth.VO_System_Severity,
    VI_RootCause := fbSystemHealth.VO_Root_Cause,
    VI_Status_Msg := fbStateManager.VO_Status_Msg
);

fbFaultLogger(
    VI_Severity := fbSystemHealth.VO_System_Severity,
    VI_RootCause := fbSystemHealth.VO_Root_Cause,
    VI_Time_MS := GVL_STATUS.G_System_Time_MS
);

GVL_STATUS.G_System_Mode_Msg := fbStateManager.VO_Status_Msg;

GVL_STATUS.G_Diagnostics.Sensor_Fault :=
    GVL_STATE.G_Heating_Sensor_Fault OR
    GVL_STATE.G_DHW_Sensor_Fault OR
    GVL_STATUS.G_Diagnostics.Manifold_Pressure_Fault_Active OR
    GVL_STATUS.G_Diagnostics.Manifold_Current_Fault_Active OR
    GVL_STATUS.G_Diagnostics.Manifold_Return_Temp_Fault_Active;

GVL_STATUS.G_Diagnostics.IO_Offline :=
    GVL_STATE.G_Heating_IO_Fault OR
    GVL_STATE.G_DHW_IO_Fault OR
    GVL_STATE.G_Ventilation_IO_Fault OR
    GVL_STATE.G_Lighting_IO_Fault;

GVL_STATUS.G_Diagnostics.Subsystem_Degraded :=
    GVL_STATE.G_Heating_Subsystem_Degraded OR
    GVL_STATE.G_DHW_Subsystem_Degraded OR
    GVL_STATE.G_Ventilation_Subsystem_Degraded OR
    GVL_STATUS.G_Diagnostics.Manifold_Pressure_Fault_Active OR
    GVL_STATUS.G_Diagnostics.Manifold_Current_Fault_Active OR
    GVL_STATUS.G_Diagnostics.Manifold_Return_Temp_Fault_Active;

GVL_GATEWAY.G_Gateway_HMI_Status_Message := fbHMIInterface.VO_HMI_Status_Text;
IF fbFaultLogger.VO_Last_Event_Text <> '' THEN
    GVL_HEALTH_BRIDGE.G_Last_Fault_Event_Text := fbFaultLogger.VO_Last_Event_Text;
END_IF;

GVL_STATE.G_System_Mode := fbStateManager.VO_System_Mode;

CASE GVL_STATE.G_System_Mode OF
    E_System_Operating_Mode.MODE_SAFE_STOP:
        GVL_STATE.G_System_Mode_Text := 'SAFE_STOP';

    E_System_Operating_Mode.MODE_FREEZE_PROTECTION:
        GVL_STATE.G_System_Mode_Text := 'FREEZE_PROTECTION';

    E_System_Operating_Mode.MODE_DEGRADED:
        GVL_STATE.G_System_Mode_Text := 'DEGRADED';

    ELSE
        GVL_STATE.G_System_Mode_Text := 'NORMAL';
END_CASE;

CASE fbSystemHealth.VO_Root_Cause OF
    E_System_Root_Cause.ROOT_FIRE:
        GVL_STATUS.G_System_Mode_Cause := 'Пожар/дым';
    E_System_Root_Cause.ROOT_GAS_LEAK:
        GVL_STATUS.G_System_Mode_Cause := 'Утечка газа';
    E_System_Root_Cause.ROOT_CO_CRITICAL:
        GVL_STATUS.G_System_Mode_Cause := 'Критический CO';
    E_System_Root_Cause.ROOT_CO_WARNING:
        GVL_STATUS.G_System_Mode_Cause := 'Повышенный CO';
    E_System_Root_Cause.ROOT_WATER_LEAK:
        GVL_STATUS.G_System_Mode_Cause := 'Протечка воды';
    E_System_Root_Cause.ROOT_WATCHDOG_FAULT:
        GVL_STATUS.G_System_Mode_Cause := 'Ошибка watchdog';
    E_System_Root_Cause.ROOT_IO_OFFLINE:
        GVL_STATUS.G_System_Mode_Cause := 'Недоступен модуль IO';
    E_System_Root_Cause.ROOT_COMM_FAULT:
        GVL_STATUS.G_System_Mode_Cause := 'Ошибка связи';
    E_System_Root_Cause.ROOT_SENSOR_FAULT:
        GVL_STATUS.G_System_Mode_Cause := 'Ошибка датчика';
    E_System_Root_Cause.ROOT_SUBSYSTEM_FAULT:
        GVL_STATUS.G_System_Mode_Cause := 'Ошибка подсистемы';
    ELSE
        GVL_STATUS.G_System_Mode_Cause := 'Аварийные режимы отсутствуют';
END_CASE;

VO_First_Fault_Active := fbSystemHealth.VO_First_Fault_Active;
VO_First_Fault_Type := fbSystemHealth.VO_First_Fault_Type;
VO_First_Fault_Source := fbSystemHealth.VO_First_Fault_Source;
VO_System_Severity := fbSystemHealth.VO_System_Severity;
VO_Root_Cause := fbSystemHealth.VO_Root_Cause;
VO_Watchdog_Fault := fbWatchdog.VO_Watchdog_Fault;

GVL_STATUS.G_System_Mode_Msg := fbStateManager.VO_Status_Msg;

// >>> BULK_SYNC_ANCHOR: FB_System_Health_Orchestrator <<<
END_FUNCTION_BLOCK

(* ---- FB_System_Persist_Manager.st ---- *)
// ==============================================================================
// System persist manager helper
//
// Internal helper for PRG_System.
// Owns persistent snapshot packing, controlled NVRAM write gating,
// FB_NVRAM_Manager call, and last-written buffer tracking.
// ==============================================================================
FUNCTION_BLOCK FB_System_Persist_Manager
VAR_INPUT
    VI_System_Time_MS : UDINT;
    VI_IsActivePLC : BOOL;
END_VAR

VAR_IN_OUT
    VIO_Persist_Buffer : ARRAY[0..4] OF BYTE;
    VIO_Last_Written_Persist_Buffer : ARRAY[0..4] OF BYTE;
    VIO_Persist_Buffer_Changed : BOOL;
    VIO_Last_Persist_Write_MS : UDINT;
    VIO_NVRAM_Cmd : BYTE;
    VIO_NVRAM_Offset : UDINT;
    VIO_NVRAM_Done : BOOL;
    VIO_NVRAM_Err : BOOL;
    VIO_NVRAM_ErrID : UDINT;
END_VAR

VAR
    fbNVRAMManager : FB_NVRAM_Manager;
END_VAR

// Pack persistent snapshot into compact byte buffer for controlled NVRAM mirroring
VIO_Persist_Buffer[0] := TO_BYTE(TO_INT(GVL_STATE.G_System_Mode));
IF GVL_PERSISTENT.P_Safety_Gas_Latched THEN
    VIO_Persist_Buffer[1] := BYTE#1;
ELSE
    VIO_Persist_Buffer[1] := BYTE#0;
END_IF;
IF GVL_PERSISTENT.P_Safety_Smoke_Latched THEN
    VIO_Persist_Buffer[2] := BYTE#1;
ELSE
    VIO_Persist_Buffer[2] := BYTE#0;
END_IF;
IF GVL_PERSISTENT.P_Safety_Leak_Latched THEN
    VIO_Persist_Buffer[3] := BYTE#1;
ELSE
    VIO_Persist_Buffer[3] := BYTE#0;
END_IF;
IF GVL_PERSISTENT.P_DHW_Heating_Active THEN
    VIO_Persist_Buffer[4] := BYTE#1;
ELSE
    VIO_Persist_Buffer[4] := BYTE#0;
END_IF;

VIO_Persist_Buffer_Changed :=
    (VIO_Persist_Buffer[0] <> VIO_Last_Written_Persist_Buffer[0]) OR
    (VIO_Persist_Buffer[1] <> VIO_Last_Written_Persist_Buffer[1]) OR
    (VIO_Persist_Buffer[2] <> VIO_Last_Written_Persist_Buffer[2]) OR
    (VIO_Persist_Buffer[3] <> VIO_Last_Written_Persist_Buffer[3]) OR
    (VIO_Persist_Buffer[4] <> VIO_Last_Written_Persist_Buffer[4]);

VIO_NVRAM_Cmd := 0;
VIO_NVRAM_Offset := 0;

IF GVL_CONFIG.G_HMI_Apply_Settings THEN
    // explicit config apply may request a controlled write
    VIO_NVRAM_Cmd := 1;
    GVL_CONFIG.G_HMI_Apply_Settings := FALSE;

ELSIF VIO_Persist_Buffer_Changed THEN
    // controlled write: no more often than once per 60 seconds
    IF (VIO_Last_Persist_Write_MS = 0) OR
       ((VI_System_Time_MS - VIO_Last_Persist_Write_MS) >= 60000) THEN
        VIO_NVRAM_Cmd := 1;
    END_IF;
END_IF;

fbNVRAMManager(
    VI_Command := VIO_NVRAM_Cmd,
    VI_Offset := VIO_NVRAM_Offset,
    VI_DataRef := VIO_Persist_Buffer[0],
    VI_DataSize := 5,
    VI_System_Time_MS := VI_System_Time_MS,
    VI_Operator_ID := 'SYSTEM',
    VI_IsActivePLC := VI_IsActivePLC,
    VI_TwoPersonConfirmation := FALSE,
    VO_Done => VIO_NVRAM_Done,
    VO_Error => VIO_NVRAM_Err,
    VO_ErrorID => VIO_NVRAM_ErrID
);

IF (VIO_NVRAM_Cmd = 1) AND VIO_NVRAM_Done AND NOT VIO_NVRAM_Err THEN
    VIO_Last_Written_Persist_Buffer[0] := VIO_Persist_Buffer[0];
    VIO_Last_Written_Persist_Buffer[1] := VIO_Persist_Buffer[1];
    VIO_Last_Written_Persist_Buffer[2] := VIO_Persist_Buffer[2];
    VIO_Last_Written_Persist_Buffer[3] := VIO_Persist_Buffer[3];
    VIO_Last_Written_Persist_Buffer[4] := VIO_Persist_Buffer[4];
    VIO_Last_Persist_Write_MS := VI_System_Time_MS;
END_IF;

// >>> BULK_SYNC_ANCHOR: FB_System_Persist_Manager <<<
END_FUNCTION_BLOCK
